LIN {X 0.054,Y -621.065,Z 312.138,A 0.000,B 0.000,C 90.000,E1 240.873} C_DIS
LIN {X 0.084,Y -617.103,Z 312.131,A 0.000,B 0.000,C 90.000,E1 239.587} C_DIS
LIN {X 0.303,Y -613.890,Z 312.125,A 0.000,B 0.000,C 90.000,E1 238.535} C_DIS
LIN {X 0.171,Y -609.063,Z 312.117,A 0.000,B 0.000,C 90.000,E1 236.993} C_DIS
LIN {X 0.075,Y -605.848,Z 312.111,A 0.000,B 0.000,C 90.000,E1 235.960} C_DIS
LIN {X 0.200,Y -600.104,Z 312.101,A 0.000,B 0.000,C 90.000,E1 234.116} C_DIS
LIN {X 0.333,Y -596.624,Z 312.095,A 0.000,B 0.000,C 90.000,E1 233.050} C_DIS
LIN {X -0.237,Y -590.243,Z 312.085,A 0.000,B 0.000,C 90.000,E1 231.251} C_DIS
LIN {X -0.144,Y -585.821,Z 312.077,A 0.000,B 0.000,C 90.000,E1 229.908} C_DIS
LIN {X -0.014,Y -580.499,Z 312.068,A 0.000,B 0.000,C 90.000,E1 228.286} C_DIS
LIN {X -0.102,Y -576.333,Z 312.061,A 0.000,B 0.000,C 90.000,E1 226.944} C_DIS
LIN {X -0.013,Y -572.939,Z 312.055,A 0.000,B 0.000,C 90.000,E1 225.850} C_DIS
LIN {X 0.018,Y -566.044,Z 312.043,A 0.000,B 0.000,C 90.000,E1 223.662} C_DIS
LIN {X 0.033,Y -561.867,Z 312.035,A 0.000,B 0.000,C 90.000,E1 222.285} C_DIS
LIN {X 0.080,Y -556.813,Z 312.026,A 0.000,B 0.000,C 90.000,E1 220.620} C_DIS
LIN {X -0.048,Y -552.562,Z 312.018,A 0.000,B 0.000,C 90.000,E1 219.241} C_DIS
LIN {X -0.129,Y -547.540,Z 312.009,A 0.000,B 0.000,C 90.000,E1 217.569} C_DIS
LIN {X 0.085,Y -543.291,Z 312.001,A 0.000,B 0.000,C 90.000,E1 216.137} C_DIS
LIN {X 0.077,Y -537.670,Z 311.990,A 0.000,B 0.000,C 90.000,E1 214.151} C_DIS
LIN {X -0.197,Y -533.791,Z 311.982,A 0.000,B 0.000,C 90.000,E1 212.752} C_DIS
LIN {X 0.071,Y -529.978,Z 311.974,A 0.000,B 0.000,C 90.000,E1 211.288} C_DIS
LIN {X 0.227,Y -525.621,Z 311.964,A 0.000,B 0.000,C 90.000,E1 209.539} C_DIS
LIN {X 0.147,Y -520.586,Z 311.953,A 0.000,B 0.000,C 90.000,E1 207.513} C_DIS
LIN {X 0.137,Y -517.085,Z 311.945,A 0.000,B 0.000,C 90.000,E1 206.052} C_DIS
LIN {X -0.273,Y -513.125,Z 311.935,A 0.000,B 0.000,C 90.000,E1 204.335} C_DIS
LIN {X 0.154,Y -509.144,Z 311.925,A 0.000,B 0.000,C 90.000,E1 202.514} C_DIS
LIN {X 0.007,Y -506.002,Z 311.917,A 0.000,B 0.000,C 90.000,E1 201.046} C_DIS
LIN {X -0.110,Y -502.294,Z 311.907,A 0.000,B 0.000,C 90.000,E1 199.268} C_DIS
LIN {X 0.051,Y -498.120,Z 311.895,A 0.000,B 0.000,C 90.000,E1 197.149} C_DIS
LIN {X -0.226,Y -494.818,Z 311.885,A 0.000,B 0.000,C 90.000,E1 195.371} C_DIS
LIN {X 0.189,Y -490.358,Z 311.870,A 0.000,B 0.000,C 90.000,E1 192.591} C_DIS
LIN {X -0.109,Y -486.945,Z 311.858,A 0.000,B 0.000,C 90.000,E1 190.489} C_DIS
LIN {X 0.109,Y -484.279,Z 311.848,A 0.000,B 0.000,C 90.000,E1 188.624} C_DIS
LIN {X -0.030,Y -481.304,Z 311.836,A 0.000,B 0.000,C 90.000,E1 186.486} C_DIS
LIN {X 0.219,Y -479.780,Z 311.829,A 0.000,B 0.000,C 90.000,E1 185.220} C_DIS
LIN {X 0.137,Y -476.898,Z 311.815,A 0.000,B 0.000,C 90.000,E1 182.751} C_DIS
LIN {X -0.189,Y -475.590,Z 311.809,A 0.000,B 0.000,C 90.000,E1 181.547} C_DIS
LIN {X -0.126,Y -472.809,Z 311.789,A 0.000,B 0.000,C 90.000,E1 178.108} C_DIS
LIN {X 0.151,Y -471.024,Z 311.769,A 0.000,B 0.000,C 90.000,E1 174.318} C_DIS
LIN {X -0.083,Y -470.413,Z 311.755,A 0.000,B 0.000,C 90.000,E1 171.837} C_DIS
LIN {X 0.080,Y -470.402,Z 311.739,A 0.000,B 0.000,C 90.000,E1 168.993} C_DIS
LIN {X -0.150,Y -470.751,Z 311.727,A 0.000,B 0.000,C 90.000,E1 166.825} C_DIS
LIN {X 0.079,Y -471.940,Z 311.711,A 0.000,B 0.000,C 90.000,E1 163.976} C_DIS
LIN {X -0.195,Y -473.286,Z 311.699,A 0.000,B 0.000,C 90.000,E1 161.819} C_DIS
LIN {X 0.260,Y -475.302,Z 311.683,A 0.000,B 0.000,C 90.000,E1 158.954} C_DIS
LIN {X 0.052,Y -478.623,Z 311.666,A 0.000,B 0.000,C 90.000,E1 155.869} C_DIS
LIN {X 0.114,Y -482.384,Z 311.651,A 0.000,B 0.000,C 90.000,E1 153.076} C_DIS
LIN {X -0.095,Y -486.412,Z 311.637,A 0.000,B 0.000,C 90.000,E1 150.639} C_DIS
LIN {X -0.173,Y -491.133,Z 311.623,A 0.000,B 0.000,C 90.000,E1 148.201} C_DIS
LIN {X 0.279,Y -494.405,Z 311.615,A 0.000,B 0.000,C 90.000,E1 146.628} C_DIS
LIN {X -0.166,Y -499.078,Z 311.603,A 0.000,B 0.000,C 90.000,E1 144.562} C_DIS
LIN {X -0.091,Y -502.259,Z 311.595,A 0.000,B 0.000,C 90.000,E1 143.050} C_DIS
LIN {X 0.049,Y -505.282,Z 311.586,A 0.000,B 0.000,C 90.000,E1 141.537} C_DIS
LIN {X -0.054,Y -507.425,Z 311.580,A 0.000,B 0.000,C 90.000,E1 140.356} C_DIS
LIN {X -0.131,Y -509.353,Z 311.573,A 0.000,B 0.000,C 90.000,E1 139.175} C_DIS
LIN {X 0.247,Y -510.541,Z 311.568,A 0.000,B 0.000,C 90.000,E1 138.243} C_DIS
LIN {X -0.081,Y -511.546,Z 311.563,A 0.000,B 0.000,C 90.000,E1 137.391} C_DIS
LIN {X -0.145,Y -512.482,Z 311.557,A 0.000,B 0.000,C 90.000,E1 136.215} C_DIS
LIN {X 0.161,Y -512.869,Z 311.550,A 0.000,B 0.000,C 90.000,E1 135.000} C_DIS
LIN {X -0.254,Y -512.798,Z 311.544,A 0.000,B 0.000,C 90.000,E1 133.866} C_DIS
LIN {X -0.302,Y -512.292,Z 311.537,A 0.000,B 0.000,C 90.000,E1 132.690} C_DIS
LIN {X 0.113,Y -511.580,Z 311.532,A 0.000,B 0.000,C 90.000,E1 131.757} C_DIS
LIN {X -0.205,Y -510.652,Z 311.527,A 0.000,B 0.000,C 90.000,E1 130.906} C_DIS
LIN {X -0.239,Y -509.147,Z 311.521,A 0.000,B 0.000,C 90.000,E1 129.725} C_DIS
LIN {X -0.071,Y -507.131,Z 311.512,A 0.000,B 0.000,C 90.000,E1 128.222} C_DIS
LIN {X 0.135,Y -505.013,Z 311.504,A 0.000,B 0.000,C 90.000,E1 126.710} C_DIS
LIN {X 0.113,Y -503.165,Z 311.497,A 0.000,B 0.000,C 90.000,E1 125.518} C_DIS
LIN {X -0.055,Y -500.467,Z 311.489,A 0.000,B 0.000,C 90.000,E1 124.040} C_DIS
LIN {X -0.138,Y -497.552,Z 311.481,A 0.000,B 0.000,C 90.000,E1 122.546} C_DIS
LIN {X -0.123,Y -495.184,Z 311.474,A 0.000,B 0.000,C 90.000,E1 121.337} C_DIS
LIN {X 0.118,Y -492.114,Z 311.466,A 0.000,B 0.000,C 90.000,E1 119.795} C_DIS
LIN {X 0.301,Y -487.796,Z 311.454,A 0.000,B 0.000,C 90.000,E1 117.641} C_DIS
LIN {X -0.080,Y -484.713,Z 311.445,A 0.000,B 0.000,C 90.000,E1 116.155} C_DIS
LIN {X 0.143,Y -481.605,Z 311.437,A 0.000,B 0.000,C 90.000,E1 114.591} C_DIS
LIN {X -0.125,Y -478.497,Z 311.428,A 0.000,B 0.000,C 90.000,E1 113.078} C_DIS
LIN {X -0.220,Y -474.768,Z 311.418,A 0.000,B 0.000,C 90.000,E1 111.227} C_DIS
LIN {X 0.038,Y -471.128,Z 311.407,A 0.000,B 0.000,C 90.000,E1 109.322} C_DIS
LIN {X 0.082,Y -466.328,Z 311.393,A 0.000,B 0.000,C 90.000,E1 106.804} C_DIS
LIN {X -0.163,Y -464.954,Z 311.389,A 0.000,B 0.000,C 90.000,E1 106.079} C_DIS
LIN {X -0.202,Y -464.952,Z 311.389,A 0.000,B 0.000,C 90.000,E1 106.079} C_DIS
LIN {X 0.165,Y -467.726,Z 311.383,A 0.000,B 0.000,C 90.000,E1 104.898} C_DIS
LIN {X 0.137,Y -475.934,Z 311.357,A 0.000,B 0.000,C 90.000,E1 100.197} C_DIS
LIN {X -0.024,Y -476.364,Z 311.355,A 0.000,B 0.000,C 90.000,E1 99.905} C_DIS
LIN {X -0.068,Y -481.890,Z 311.331,A 0.000,B 0.000,C 90.000,E1 95.568} C_DIS
LIN {X -0.220,Y -482.197,Z 311.329,A 0.000,B 0.000,C 90.000,E1 95.277} C_DIS
LIN {X 0.198,Y -485.374,Z 311.305,A 0.000,B 0.000,C 90.000,E1 90.917} C_DIS
LIN {X 0.023,Y -485.531,Z 311.304,A 0.000,B 0.000,C 90.000,E1 90.630} C_DIS
LIN {X 0.230,Y -486.350,Z 311.281,A 0.000,B 0.000,C 90.000,E1 86.617} C_DIS
LIN {X 0.055,Y -486.369,Z 311.280,A 0.000,B 0.000,C 90.000,E1 86.331} C_DIS
LIN {X 0.223,Y -486.057,Z 311.276,A 0.000,B 0.000,C 90.000,E1 85.698} C_DIS
LIN {X 0.079,Y -484.693,Z 311.254,A 0.000,B 0.000,C 90.000,E1 81.724} C_DIS
LIN {X -0.053,Y -484.524,Z 311.252,A 0.000,B 0.000,C 90.000,E1 81.432} C_DIS
LIN {X -0.183,Y -480.460,Z 311.227,A 0.000,B 0.000,C 90.000,E1 76.825} C_DIS
LIN {X -0.138,Y -475.986,Z 311.210,A 0.000,B 0.000,C 90.000,E1 73.740} C_DIS
LIN {X 0.178,Y -480.585,Z 311.199,A 0.000,B 0.000,C 90.000,E1 71.819} C_DIS
LIN {X -0.159,Y -485.320,Z 311.189,A 0.000,B 0.000,C 90.000,E1 70.007} C_DIS
LIN {X -0.080,Y -489.458,Z 311.180,A 0.000,B 0.000,C 90.000,E1 68.465} C_DIS
LIN {X 0.044,Y -492.837,Z 311.174,A 0.000,B 0.000,C 90.000,E1 67.230} C_DIS
LIN {X -0.191,Y -497.106,Z 311.165,A 0.000,B 0.000,C 90.000,E1 65.741} C_DIS
LIN {X -0.253,Y -503.092,Z 311.153,A 0.000,B 0.000,C 90.000,E1 63.640} C_DIS
LIN {X 0.123,Y -507.432,Z 311.145,A 0.000,B 0.000,C 90.000,E1 62.103} C_DIS
LIN {X 0.017,Y -512.604,Z 311.135,A 0.000,B 0.000,C 90.000,E1 60.333} C_DIS
LIN {X -0.080,Y -516.937,Z 311.127,A 0.000,B 0.000,C 90.000,E1 58.869} C_DIS
LIN {X -0.162,Y -522.069,Z 311.117,A 0.000,B 0.000,C 90.000,E1 57.120} C_DIS
LIN {X -0.252,Y -526.246,Z 311.109,A 0.000,B 0.000,C 90.000,E1 55.674} C_DIS
LIN {X 0.034,Y -530.220,Z 311.101,A 0.000,B 0.000,C 90.000,E1 54.196} C_DIS
LIN {X -0.023,Y -533.243,Z 311.095,A 0.000,B 0.000,C 90.000,E1 53.050} C_DIS
LIN {X -0.039,Y -535.952,Z 311.088,A 0.000,B 0.000,C 90.000,E1 51.904} C_DIS
LIN {X 0.318,Y -538.475,Z 311.082,A 0.000,B 0.000,C 90.000,E1 50.723} C_DIS
LIN {X -0.077,Y -539.629,Z 311.079,A 0.000,B 0.000,C 90.000,E1 50.194} C_DIS
LIN {X -0.062,Y -542.242,Z 311.071,A 0.000,B 0.000,C 90.000,E1 48.771} C_DIS
LIN {X -0.050,Y -543.727,Z 311.066,A 0.000,B 0.000,C 90.000,E1 47.919} C_DIS
LIN {X -0.022,Y -544.977,Z 311.062,A 0.000,B 0.000,C 90.000,E1 47.067} C_DIS
LIN {X 0.043,Y -546.765,Z 311.054,A 0.000,B 0.000,C 90.000,E1 45.648} C_DIS
LIN {X -0.293,Y -547.576,Z 311.049,A 0.000,B 0.000,C 90.000,E1 44.838} C_DIS
LIN {X 0.194,Y -548.560,Z 311.041,A 0.000,B 0.000,C 90.000,E1 43.380} C_DIS
LIN {X -0.095,Y -549.162,Z 311.035,A 0.000,B 0.000,C 90.000,E1 42.285} C_DIS
LIN {X 0.081,Y -549.559,Z 311.027,A 0.000,B 0.000,C 90.000,E1 40.862} C_DIS
LIN {X 0.168,Y -549.577,Z 311.022,A 0.000,B 0.000,C 90.000,E1 40.011} C_DIS
LIN {X -0.049,Y -549.318,Z 311.016,A 0.000,B 0.000,C 90.000,E1 38.910} C_DIS
LIN {X -0.321,Y -548.907,Z 311.012,A 0.000,B 0.000,C 90.000,E1 38.096} C_DIS
LIN {X -0.063,Y -547.928,Z 311.004,A 0.000,B 0.000,C 90.000,E1 36.664} C_DIS
LIN {X 0.129,Y -546.952,Z 310.997,A 0.000,B 0.000,C 90.000,E1 35.518} C_DIS
LIN {X 0.027,Y -545.669,Z 310.990,A 0.000,B 0.000,C 90.000,E1 34.119} C_DIS
LIN {X 0.056,Y -544.321,Z 310.982,A 0.000,B 0.000,C 90.000,E1 32.704} C_DIS
LIN {X -0.159,Y -542.194,Z 310.969,A 0.000,B 0.000,C 90.000,E1 30.463} C_DIS
LIN {X -0.260,Y -540.386,Z 310.958,A 0.000,B 0.000,C 90.000,E1 28.487} C_DIS
LIN {X -0.111,Y -539.313,Z 310.952,A 0.000,B 0.000,C 90.000,E1 27.334} C_DIS
LIN {X -0.007,Y -537.941,Z 310.944,A 0.000,B 0.000,C 90.000,E1 25.899} C_DIS
LIN {X -0.193,Y -536.382,Z 310.934,A 0.000,B 0.000,C 90.000,E1 24.207} C_DIS
LIN {X -0.199,Y -534.694,Z 310.923,A 0.000,B 0.000,C 90.000,E1 22.206} C_DIS
LIN {X -0.069,Y -533.850,Z 310.917,A 0.000,B 0.000,C 90.000,E1 21.046} C_DIS
LIN {X 0.165,Y -532.393,Z 310.904,A 0.000,B 0.000,C 90.000,E1 18.725} C_DIS
LIN {X 0.189,Y -531.050,Z 310.890,A 0.000,B 0.000,C 90.000,E1 16.134} C_DIS
LIN {X 0.178,Y -530.305,Z 310.879,A 0.000,B 0.000,C 90.000,E1 14.120} C_DIS
LIN {X 0.023,Y -529.791,Z 310.867,A 0.000,B 0.000,C 90.000,E1 12.119} C_DIS
LIN {X 0.202,Y -529.576,Z 310.855,A 0.000,B 0.000,C 90.000,E1 9.792} C_DIS
LIN {X -0.192,Y -529.790,Z 310.840,A 0.000,B 0.000,C 90.000,E1 7.239} C_DIS
LIN {X -0.217,Y -530.398,Z 310.827,A 0.000,B 0.000,C 90.000,E1 4.935} C_DIS
LIN {X -0.264,Y -531.101,Z 310.818,A 0.000,B 0.000,C 90.000,E1 3.212} C_DIS
LIN {X 0.227,Y -532.011,Z 310.808,A 0.000,B 0.000,C 90.000,E1 1.432} C_DIS
LIN {X 0.189,Y -533.352,Z 310.796,A 0.000,B 0.000,C 90.000,E1 359.198} C_DIS
LIN {X 0.175,Y -535.039,Z 310.785,A 0.000,B 0.000,C 90.000,E1 357.192} C_DIS
LIN {X 0.229,Y -536.424,Z 310.777,A 0.000,B 0.000,C 90.000,E1 355.755} C_DIS
LIN {X -0.060,Y -539.508,Z 310.761,A 0.000,B 0.000,C 90.000,E1 352.932} C_DIS
LIN {X 0.205,Y -542.803,Z 310.750,A 0.000,B 0.000,C 90.000,E1 350.914} C_DIS
LIN {X 0.248,Y -549.753,Z 310.731,A 0.000,B 0.000,C 90.000,E1 347.521} C_DIS
LIN {X -0.151,Y -554.083,Z 310.722,A 0.000,B 0.000,C 90.000,E1 345.880} C_DIS
LIN {X 0.231,Y -560.124,Z 310.709,A 0.000,B 0.000,C 90.000,E1 343.614} C_DIS
LIN {X -0.212,Y -564.870,Z 310.700,A 0.000,B 0.000,C 90.000,E1 342.000} C_DIS
LIN {X 0.143,Y -569.679,Z 310.691,A 0.000,B 0.000,C 90.000,E1 340.315} C_DIS
LIN {X 0.299,Y -571.368,Z 310.688,A 0.000,B 0.000,C 90.000,E1 339.752} C_DIS
LIN {X 0.095,Y -573.791,Z 310.683,A 0.000,B 0.000,C 90.000,E1 338.954} C_DIS
LIN {X 0.291,Y -577.312,Z 310.677,A 0.000,B 0.000,C 90.000,E1 337.847} C_DIS
LIN {X -0.002,Y -580.918,Z 310.671,A 0.000,B 0.000,C 90.000,E1 336.794} C_DIS
LIN {X 0.148,Y -585.383,Z 310.664,A 0.000,B 0.000,C 90.000,E1 335.433} C_DIS
LIN {X -0.135,Y -592.066,Z 310.653,A 0.000,B 0.000,C 90.000,E1 333.589} C_DIS
LIN {X 0.092,Y -597.745,Z 310.644,A 0.000,B 0.000,C 90.000,E1 331.975} C_DIS
LIN {X -0.018,Y -602.312,Z 310.637,A 0.000,B 0.000,C 90.000,E1 330.667} C_DIS
LIN {X 0.192,Y -607.892,Z 310.628,A 0.000,B 0.000,C 90.000,E1 329.076} C_DIS
LIN {X 0.278,Y -614.299,Z 310.618,A 0.000,B 0.000,C 90.000,E1 327.248} C_DIS
LIN {X 0.273,Y -617.854,Z 310.612,A 0.000,B 0.000,C 90.000,E1 326.215} C_DIS
LIN {X -0.228,Y -622.276,Z 310.605,A 0.000,B 0.000,C 90.000,E1 324.975} C_DIS
LIN {X -0.110,Y -624.819,Z 310.601,A 0.000,B 0.000,C 90.000,E1 324.196} C_DIS
LIN {X 0.386,Y -628.014,Z 310.595,A 0.000,B 0.000,C 90.000,E1 323.130} C_DIS
LIN {X -0.099,Y -631.744,Z 310.588,A 0.000,B 0.000,C 90.000,E1 321.904} C_DIS
LIN {X 0.246,Y -636.116,Z 310.580,A 0.000,B 0.000,C 90.000,E1 320.356} C_DIS
LIN {X 0.193,Y -640.561,Z 310.572,A 0.000,B 0.000,C 90.000,E1 318.852} C_DIS
LIN {X -0.103,Y -643.426,Z 310.566,A 0.000,B 0.000,C 90.000,E1 317.877} C_DIS
LIN {X -0.308,Y -650.814,Z 310.552,A 0.000,B 0.000,C 90.000,E1 315.405} C_DIS
LIN {X -0.047,Y -653.782,Z 310.547,A 0.000,B 0.000,C 90.000,E1 314.393} C_DIS
LIN {X -0.225,Y -657.191,Z 310.540,A 0.000,B 0.000,C 90.000,E1 313.176} C_DIS
LIN {X 0.113,Y -660.442,Z 310.533,A 0.000,B 0.000,C 90.000,E1 311.919} C_DIS
LIN {X -0.398,Y -662.295,Z 310.529,A 0.000,B 0.000,C 90.000,E1 311.229} C_DIS
LIN {X 0.022,Y -664.597,Z 310.523,A 0.000,B 0.000,C 90.000,E1 310.216} C_DIS
LIN {X 0.115,Y -667.184,Z 310.517,A 0.000,B 0.000,C 90.000,E1 308.991} C_DIS
LIN {X 0.165,Y -669.104,Z 310.511,A 0.000,B 0.000,C 90.000,E1 308.016} C_DIS
LIN {X -0.165,Y -670.398,Z 310.507,A 0.000,B 0.000,C 90.000,E1 307.317} C_DIS
LIN {X -0.093,Y -671.847,Z 310.502,A 0.000,B 0.000,C 90.000,E1 306.343} C_DIS
LIN {X -0.258,Y -673.002,Z 310.497,A 0.000,B 0.000,C 90.000,E1 305.391} C_DIS
LIN {X 0.396,Y -673.569,Z 310.493,A 0.000,B 0.000,C 90.000,E1 304.612} C_DIS
LIN {X 0.113,Y -673.892,Z 310.488,A 0.000,B 0.000,C 90.000,E1 303.913} C_DIS
LIN {X -0.009,Y -673.873,Z 310.483,A 0.000,B 0.000,C 90.000,E1 302.959} C_DIS
LIN {X 0.275,Y -673.725,Z 310.479,A 0.000,B 0.000,C 90.000,E1 302.212} C_DIS
LIN {X -0.019,Y -673.187,Z 310.475,A 0.000,B 0.000,C 90.000,E1 301.514} C_DIS
LIN {X -0.096,Y -672.317,Z 310.471,A 0.000,B 0.000,C 90.000,E1 300.797} C_DIS
LIN {X 0.328,Y -670.772,Z 310.466,A 0.000,B 0.000,C 90.000,E1 299.795} C_DIS
LIN {X 0.236,Y -669.265,Z 310.462,A 0.000,B 0.000,C 90.000,E1 299.077} C_DIS
LIN {X -0.143,Y -666.552,Z 310.455,A 0.000,B 0.000,C 90.000,E1 297.897} C_DIS
LIN {X 0.016,Y -663.590,Z 310.448,A 0.000,B 0.000,C 90.000,E1 296.668} C_DIS
LIN {X -0.167,Y -660.470,Z 310.441,A 0.000,B 0.000,C 90.000,E1 295.463} C_DIS
LIN {X 0.198,Y -657.146,Z 310.435,A 0.000,B 0.000,C 90.000,E1 294.207} C_DIS
LIN {X -0.243,Y -653.100,Z 310.426,A 0.000,B 0.000,C 90.000,E1 292.770} C_DIS
LIN {X -0.194,Y -651.088,Z 310.422,A 0.000,B 0.000,C 90.000,E1 292.025} C_DIS
LIN {X -0.163,Y -647.115,Z 310.414,A 0.000,B 0.000,C 90.000,E1 290.536} C_DIS
LIN {X -0.164,Y -642.085,Z 310.403,A 0.000,B 0.000,C 90.000,E1 288.544} C_DIS
LIN {X -0.197,Y -635.149,Z 310.386,A 0.000,B 0.000,C 90.000,E1 285.536} C_DIS
LIN {X -0.172,Y -630.235,Z 310.372,A 0.000,B 0.000,C 90.000,E1 283.008} C_DIS
LIN {X -0.215,Y -625.615,Z 310.355,A 0.000,B 0.000,C 90.000,E1 279.962} C_DIS
LIN {X 0.000,Y -622.967,Z 310.343,A 0.000,B 0.000,C 90.000,E1 277.644} C_DIS
LIN {X 0.053,Y -621.061,Z 310.330,A 0.000,B 0.000,C 90.000,E1 275.334} C_DIS
LIN {X 0.244,Y -619.846,Z 310.315,A 0.000,B 0.000,C 90.000,E1 272.751} C_DIS
LIN {X 0.052,Y -619.395,Z 310.300,A 0.000,B 0.000,C 90.000,E1 269.943} C_DIS
LIN {X 0.173,Y -620.108,Z 310.283,A 0.000,B 0.000,C 90.000,E1 266.849} C_DIS
LIN {X -0.271,Y -621.277,Z 310.271,A 0.000,B 0.000,C 90.000,E1 264.837} C_DIS
LIN {X 0.007,Y -622.958,Z 310.260,A 0.000,B 0.000,C 90.000,E1 262.761} C_DIS
LIN {X 0.195,Y -625.348,Z 310.247,A 0.000,B 0.000,C 90.000,E1 260.443} C_DIS
LIN {X 0.145,Y -627.977,Z 310.236,A 0.000,B 0.000,C 90.000,E1 258.409} C_DIS
LIN {X -0.201,Y -630.937,Z 310.224,A 0.000,B 0.000,C 90.000,E1 256.408} C_DIS
LIN {X 0.058,Y -633.131,Z 310.216,A 0.000,B 0.000,C 90.000,E1 254.866} C_DIS
LIN {X 0.302,Y -633.774,Z 310.213,A 0.000,B 0.000,C 90.000,E1 254.338} C_DIS
LIN {X 0.178,Y -634.938,Z 310.206,A 0.000,B 0.000,C 90.000,E1 253.087} C_DIS
LIN {X -0.360,Y -635.842,Z 310.201,A 0.000,B 0.000,C 90.000,E1 252.127} C_DIS
LIN {X -0.082,Y -636.461,Z 310.195,A 0.000,B 0.000,C 90.000,E1 251.094} C_DIS
LIN {X 0.178,Y -636.676,Z 310.191,A 0.000,B 0.000,C 90.000,E1 250.315} C_DIS
LIN {X -0.133,Y -636.627,Z 310.185,A 0.000,B 0.000,C 90.000,E1 249.337} C_DIS
LIN {X -0.251,Y -636.412,Z 310.181,A 0.000,B 0.000,C 90.000,E1 248.592} C_DIS
LIN {X 0.263,Y -635.595,Z 310.175,A 0.000,B 0.000,C 90.000,E1 247.539} C_DIS
LIN {X 0.098,Y -635.033,Z 310.173,A 0.000,B 0.000,C 90.000,E1 247.050} C_DIS
LIN {X 0.181,Y -634.369,Z 310.170,A 0.000,B 0.000,C 90.000,E1 246.538} C_DIS
LIN {X 0.045,Y -633.128,Z 310.166,A 0.000,B 0.000,C 90.000,E1 245.793} C_DIS
LIN {X 0.121,Y -632.218,Z 310.163,A 0.000,B 0.000,C 90.000,E1 245.281} C_DIS
LIN {X -0.043,Y -630.586,Z 310.159,A 0.000,B 0.000,C 90.000,E1 244.537} C_DIS
LIN {X 0.071,Y -628.088,Z 310.153,A 0.000,B 0.000,C 90.000,E1 243.512} C_DIS
LIN {X 0.151,Y -625.236,Z 310.147,A 0.000,B 0.000,C 90.000,E1 242.487} C_DIS
LIN {X -0.358,Y -621.437,Z 310.140,A 0.000,B 0.000,C 90.000,E1 241.257} C_DIS
LIN {X -0.093,Y -617.580,Z 310.133,A 0.000,B 0.000,C 90.000,E1 239.950} C_DIS
LIN {X -0.114,Y -613.641,Z 310.126,A 0.000,B 0.000,C 90.000,E1 238.663} C_DIS
LIN {X -0.243,Y -608.795,Z 310.117,A 0.000,B 0.000,C 90.000,E1 237.120} C_DIS
LIN {X -0.337,Y -605.632,Z 310.111,A 0.000,B 0.000,C 90.000,E1 236.087} C_DIS
LIN {X -0.221,Y -601.541,Z 310.104,A 0.000,B 0.000,C 90.000,E1 234.769} C_DIS
LIN {X -0.313,Y -599.112,Z 310.100,A 0.000,B 0.000,C 90.000,E1 233.989} C_DIS
LIN {X -0.194,Y -595.564,Z 310.094,A 0.000,B 0.000,C 90.000,E1 232.924} C_DIS
LIN {X 0.037,Y -589.256,Z 310.084,A 0.000,B 0.000,C 90.000,E1 231.045} C_DIS
LIN {X 0.106,Y -584.857,Z 310.076,A 0.000,B 0.000,C 90.000,E1 229.703} C_DIS
LIN {X 0.208,Y -579.597,Z 310.067,A 0.000,B 0.000,C 90.000,E1 228.081} C_DIS
LIN {X 0.068,Y -575.454,Z 310.060,A 0.000,B 0.000,C 90.000,E1 226.743} C_DIS
LIN {X 0.152,Y -572.042,Z 310.054,A 0.000,B 0.000,C 90.000,E1 225.648} C_DIS
LIN {X -0.335,Y -566.078,Z 310.043,A 0.000,B 0.000,C 90.000,E1 223.785} C_DIS
LIN {X 0.090,Y -561.927,Z 310.035,A 0.000,B 0.000,C 90.000,E1 222.366} C_DIS
LIN {X 0.058,Y -557.749,Z 310.028,A 0.000,B 0.000,C 90.000,E1 220.987} C_DIS
LIN {X 0.020,Y -553.531,Z 310.020,A 0.000,B 0.000,C 90.000,E1 219.600} C_DIS
LIN {X -0.114,Y -548.496,Z 310.011,A 0.000,B 0.000,C 90.000,E1 217.935} C_DIS
LIN {X 0.119,Y -544.254,Z 310.003,A 0.000,B 0.000,C 90.000,E1 216.503} C_DIS
LIN {X 0.011,Y -537.756,Z 309.990,A 0.000,B 0.000,C 90.000,E1 214.246} C_DIS
LIN {X 0.180,Y -534.636,Z 309.984,A 0.000,B 0.000,C 90.000,E1 213.086} C_DIS
LIN {X 0.131,Y -529.207,Z 309.973,A 0.000,B 0.000,C 90.000,E1 211.082} C_DIS
LIN {X 0.265,Y -524.860,Z 309.963,A 0.000,B 0.000,C 90.000,E1 209.333} C_DIS
LIN {X -0.079,Y -519.798,Z 309.952,A 0.000,B 0.000,C 90.000,E1 207.334} C_DIS
LIN {X 0.131,Y -516.279,Z 309.944,A 0.000,B 0.000,C 90.000,E1 205.848} C_DIS
LIN {X 0.043,Y -513.004,Z 309.936,A 0.000,B 0.000,C 90.000,E1 204.387} C_DIS
LIN {X -0.100,Y -508.399,Z 309.924,A 0.000,B 0.000,C 90.000,E1 202.333} C_DIS
LIN {X -0.163,Y -504.665,Z 309.914,A 0.000,B 0.000,C 90.000,E1 200.556} C_DIS
LIN {X 0.089,Y -501.654,Z 309.906,A 0.000,B 0.000,C 90.000,E1 199.033} C_DIS
LIN {X 0.238,Y -497.600,Z 309.894,A 0.000,B 0.000,C 90.000,E1 196.913} C_DIS
LIN {X -0.196,Y -492.370,Z 309.877,A 0.000,B 0.000,C 90.000,E1 193.939} C_DIS
LIN {X -0.129,Y -489.983,Z 309.869,A 0.000,B 0.000,C 90.000,E1 192.411} C_DIS
LIN {X 0.038,Y -486.615,Z 309.857,A 0.000,B 0.000,C 90.000,E1 190.254} C_DIS
LIN {X -0.178,Y -484.454,Z 309.849,A 0.000,B 0.000,C 90.000,E1 188.746} C_DIS
LIN {X 0.182,Y -481.486,Z 309.837,A 0.000,B 0.000,C 90.000,E1 186.549} C_DIS
LIN {X -0.192,Y -479.552,Z 309.828,A 0.000,B 0.000,C 90.000,E1 185.049} C_DIS
LIN {X 0.202,Y -476.726,Z 309.814,A 0.000,B 0.000,C 90.000,E1 182.522} C_DIS
LIN {X -0.126,Y -475.405,Z 309.807,A 0.000,B 0.000,C 90.000,E1 181.318} C_DIS
LIN {X 0.148,Y -472.962,Z 309.790,A 0.000,B 0.000,C 90.000,E1 178.165} C_DIS
LIN {X 0.151,Y -471.273,Z 309.771,A 0.000,B 0.000,C 90.000,E1 174.723} C_DIS
LIN {X -0.080,Y -470.643,Z 309.757,A 0.000,B 0.000,C 90.000,E1 172.243} C_DIS
LIN {X -0.084,Y -470.520,Z 309.739,A 0.000,B 0.000,C 90.000,E1 169.106} C_DIS
LIN {X 0.188,Y -471.119,Z 309.722,A 0.000,B 0.000,C 90.000,E1 165.936} C_DIS
LIN {X 0.212,Y -472.148,Z 309.710,A 0.000,B 0.000,C 90.000,E1 163.740} C_DIS
LIN {X -0.061,Y -473.472,Z 309.698,A 0.000,B 0.000,C 90.000,E1 161.583} C_DIS
LIN {X 0.001,Y -475.046,Z 309.686,A 0.000,B 0.000,C 90.000,E1 159.390} C_DIS
LIN {X -0.142,Y -476.710,Z 309.675,A 0.000,B 0.000,C 90.000,E1 157.539} C_DIS
LIN {X -0.044,Y -478.543,Z 309.667,A 0.000,B 0.000,C 90.000,E1 155.973} C_DIS
LIN {X 0.033,Y -482.245,Z 309.651,A 0.000,B 0.000,C 90.000,E1 153.179} C_DIS
LIN {X 0.024,Y -486.208,Z 309.637,A 0.000,B 0.000,C 90.000,E1 150.717} C_DIS
LIN {X -0.234,Y -491.462,Z 309.622,A 0.000,B 0.000,C 90.000,E1 147.995} C_DIS
LIN {X 0.225,Y -494.635,Z 309.614,A 0.000,B 0.000,C 90.000,E1 146.421} C_DIS
LIN {X 0.073,Y -499.143,Z 309.602,A 0.000,B 0.000,C 90.000,E1 144.322} C_DIS
LIN {X -0.023,Y -501.622,Z 309.595,A 0.000,B 0.000,C 90.000,E1 143.130} C_DIS
LIN {X 0.103,Y -504.588,Z 309.587,A 0.000,B 0.000,C 90.000,E1 141.618} C_DIS
LIN {X -0.013,Y -506.685,Z 309.580,A 0.000,B 0.000,C 90.000,E1 140.436} C_DIS
LIN {X -0.101,Y -508.590,Z 309.574,A 0.000,B 0.000,C 90.000,E1 139.256} C_DIS
LIN {X 0.266,Y -509.757,Z 309.569,A 0.000,B 0.000,C 90.000,E1 138.324} C_DIS
LIN {X -0.069,Y -510.762,Z 309.564,A 0.000,B 0.000,C 90.000,E1 137.472} C_DIS
LIN {X -0.045,Y -511.443,Z 309.559,A 0.000,B 0.000,C 90.000,E1 136.581} C_DIS
LIN {X 0.107,Y -511.858,Z 309.556,A 0.000,B 0.000,C 90.000,E1 135.972} C_DIS
LIN {X 0.040,Y -512.129,Z 309.549,A 0.000,B 0.000,C 90.000,E1 134.798} C_DIS
LIN {X -0.279,Y -512.055,Z 309.544,A 0.000,B 0.000,C 90.000,E1 133.947} C_DIS
LIN {X 0.134,Y -511.735,Z 309.539,A 0.000,B 0.000,C 90.000,E1 133.014} C_DIS
LIN {X -0.179,Y -511.122,Z 309.534,A 0.000,B 0.000,C 90.000,E1 132.162} C_DIS
LIN {X 0.223,Y -510.290,Z 309.529,A 0.000,B 0.000,C 90.000,E1 131.229} C_DIS
LIN {X 0.028,Y -508.518,Z 309.521,A 0.000,B 0.000,C 90.000,E1 129.769} C_DIS
LIN {X -0.239,Y -506.074,Z 309.511,A 0.000,B 0.000,C 90.000,E1 128.016} C_DIS
LIN {X 0.057,Y -504.360,Z 309.504,A 0.000,B 0.000,C 90.000,E1 126.790} C_DIS
LIN {X 0.029,Y -502.503,Z 309.498,A 0.000,B 0.000,C 90.000,E1 125.598} C_DIS
LIN {X -0.025,Y -500.364,Z 309.491,A 0.000,B 0.000,C 90.000,E1 124.405} C_DIS
LIN {X -0.116,Y -498.114,Z 309.484,A 0.000,B 0.000,C 90.000,E1 123.214} C_DIS
LIN {X 0.029,Y -494.589,Z 309.474,A 0.000,B 0.000,C 90.000,E1 121.386} C_DIS
LIN {X 0.264,Y -490.887,Z 309.464,A 0.000,B 0.000,C 90.000,E1 119.539} C_DIS
LIN {X 0.182,Y -487.208,Z 309.454,A 0.000,B 0.000,C 90.000,E1 117.719} C_DIS
LIN {X -0.204,Y -484.118,Z 309.446,A 0.000,B 0.000,C 90.000,E1 116.232} C_DIS
LIN {X 0.215,Y -481.035,Z 309.437,A 0.000,B 0.000,C 90.000,E1 114.643} C_DIS
LIN {X -0.083,Y -477.301,Z 309.427,A 0.000,B 0.000,C 90.000,E1 112.823} C_DIS
LIN {X -0.158,Y -474.876,Z 309.420,A 0.000,B 0.000,C 90.000,E1 111.589} C_DIS
LIN {X -0.059,Y -471.233,Z 309.409,A 0.000,B 0.000,C 90.000,E1 109.704} C_DIS
LIN {X -0.043,Y -467.597,Z 309.399,A 0.000,B 0.000,C 90.000,E1 107.819} C_DIS
LIN {X -0.265,Y -464.685,Z 309.390,A 0.000,B 0.000,C 90.000,E1 106.205} C_DIS
LIN {X 0.142,Y -464.687,Z 309.390,A 0.000,B 0.000,C 90.000,E1 106.150} C_DIS
LIN {X 0.152,Y -467.594,Z 309.383,A 0.000,B 0.000,C 90.000,E1 104.954} C_DIS
LIN {X -0.115,Y -468.592,Z 309.380,A 0.000,B 0.000,C 90.000,E1 104.356} C_DIS
LIN {X 0.111,Y -475.823,Z 309.357,A 0.000,B 0.000,C 90.000,E1 100.254} C_DIS
LIN {X -0.052,Y -476.314,Z 309.355,A 0.000,B 0.000,C 90.000,E1 99.962} C_DIS
LIN {X -0.104,Y -481.805,Z 309.331,A 0.000,B 0.000,C 90.000,E1 95.625} C_DIS
LIN {X 0.222,Y -482.175,Z 309.330,A 0.000,B 0.000,C 90.000,E1 95.277} C_DIS
LIN {X 0.157,Y -485.319,Z 309.306,A 0.000,B 0.000,C 90.000,E1 90.974} C_DIS
LIN {X -0.018,Y -485.536,Z 309.304,A 0.000,B 0.000,C 90.000,E1 90.688} C_DIS
LIN {X 0.189,Y -486.324,Z 309.282,A 0.000,B 0.000,C 90.000,E1 86.674} C_DIS
LIN {X -0.161,Y -486.298,Z 309.278,A 0.000,B 0.000,C 90.000,E1 86.102} C_DIS
LIN {X 0.043,Y -484.695,Z 309.254,A 0.000,B 0.000,C 90.000,E1 81.781} C_DIS
LIN {X -0.089,Y -484.588,Z 309.253,A 0.000,B 0.000,C 90.000,E1 81.489} C_DIS
LIN {X -0.209,Y -480.524,Z 309.227,A 0.000,B 0.000,C 90.000,E1 76.881} C_DIS
LIN {X -0.132,Y -475.792,Z 309.209,A 0.000,B 0.000,C 90.000,E1 73.559} C_DIS
LIN {X -0.023,Y -481.353,Z 309.196,A 0.000,B 0.000,C 90.000,E1 71.275} C_DIS
LIN {X -0.129,Y -488.603,Z 309.181,A 0.000,B 0.000,C 90.000,E1 68.518} C_DIS
LIN {X 0.021,Y -492.802,Z 309.172,A 0.000,B 0.000,C 90.000,E1 66.975} C_DIS
LIN {X -0.212,Y -497.069,Z 309.164,A 0.000,B 0.000,C 90.000,E1 65.485} C_DIS
LIN {X -0.273,Y -503.050,Z 309.152,A 0.000,B 0.000,C 90.000,E1 63.384} C_DIS
LIN {X 0.025,Y -506.550,Z 309.145,A 0.000,B 0.000,C 90.000,E1 62.153} C_DIS
LIN {X -0.094,Y -511.730,Z 309.135,A 0.000,B 0.000,C 90.000,E1 60.383} C_DIS
LIN {X 0.242,Y -516.076,Z 309.127,A 0.000,B 0.000,C 90.000,E1 58.869} C_DIS
LIN {X -0.234,Y -520.331,Z 309.119,A 0.000,B 0.000,C 90.000,E1 57.454} C_DIS
LIN {X 0.039,Y -525.419,Z 309.109,A 0.000,B 0.000,C 90.000,E1 55.674} C_DIS
LIN {X 0.312,Y -529.405,Z 309.101,A 0.000,B 0.000,C 90.000,E1 54.196} C_DIS
LIN {X 0.245,Y -532.411,Z 309.095,A 0.000,B 0.000,C 90.000,E1 53.050} C_DIS
LIN {X 0.219,Y -535.126,Z 309.089,A 0.000,B 0.000,C 90.000,E1 51.904} C_DIS
LIN {X -0.193,Y -537.684,Z 309.082,A 0.000,B 0.000,C 90.000,E1 50.803} C_DIS
LIN {X -0.216,Y -540.451,Z 309.074,A 0.000,B 0.000,C 90.000,E1 49.380} C_DIS
LIN {X 0.170,Y -542.928,Z 309.066,A 0.000,B 0.000,C 90.000,E1 47.919} C_DIS
LIN {X 0.190,Y -544.258,Z 309.062,A 0.000,B 0.000,C 90.000,E1 47.067} C_DIS
LIN {X 0.242,Y -546.007,Z 309.054,A 0.000,B 0.000,C 90.000,E1 45.648} C_DIS
LIN {X 0.270,Y -546.590,Z 309.051,A 0.000,B 0.000,C 90.000,E1 45.081} C_DIS
LIN {X 0.338,Y -547.446,Z 309.044,A 0.000,B 0.000,C 90.000,E1 43.947} C_DIS
LIN {X 0.035,Y -548.181,Z 309.038,A 0.000,B 0.000,C 90.000,E1 42.852} C_DIS
LIN {X -0.256,Y -548.609,Z 309.032,A 0.000,B 0.000,C 90.000,E1 41.757} C_DIS
LIN {X -0.133,Y -548.873,Z 309.026,A 0.000,B 0.000,C 90.000,E1 40.620} C_DIS
LIN {X -0.011,Y -548.826,Z 309.019,A 0.000,B 0.000,C 90.000,E1 39.483} C_DIS
LIN {X 0.139,Y -548.587,Z 309.015,A 0.000,B 0.000,C 90.000,E1 38.624} C_DIS
LIN {X -0.140,Y -548.140,Z 309.010,A 0.000,B 0.000,C 90.000,E1 37.810} C_DIS
LIN {X 0.057,Y -547.373,Z 309.004,A 0.000,B 0.000,C 90.000,E1 36.664} C_DIS
LIN {X 0.240,Y -546.447,Z 308.997,A 0.000,B 0.000,C 90.000,E1 35.518} C_DIS
LIN {X -0.139,Y -544.929,Z 308.988,A 0.000,B 0.000,C 90.000,E1 33.865} C_DIS
LIN {X 0.177,Y -543.566,Z 308.980,A 0.000,B 0.000,C 90.000,E1 32.418} C_DIS
LIN {X -0.071,Y -541.469,Z 308.968,A 0.000,B 0.000,C 90.000,E1 30.178} C_DIS
LIN {X 0.018,Y -539.641,Z 308.957,A 0.000,B 0.000,C 90.000,E1 28.180} C_DIS
LIN {X -0.133,Y -538.024,Z 308.947,A 0.000,B 0.000,C 90.000,E1 26.488} C_DIS
LIN {X -0.152,Y -535.879,Z 308.934,A 0.000,B 0.000,C 90.000,E1 24.207} C_DIS
LIN {X 0.236,Y -533.766,Z 308.920,A 0.000,B 0.000,C 90.000,E1 21.589} C_DIS
LIN {X 0.167,Y -531.818,Z 308.904,A 0.000,B 0.000,C 90.000,E1 18.725} C_DIS
LIN {X 0.201,Y -530.306,Z 308.888,A 0.000,B 0.000,C 90.000,E1 15.843} C_DIS
LIN {X -0.272,Y -529.383,Z 308.874,A 0.000,B 0.000,C 90.000,E1 13.300} C_DIS
LIN {X 0.038,Y -529.044,Z 308.864,A 0.000,B 0.000,C 90.000,E1 11.535} C_DIS
LIN {X 0.133,Y -528.857,Z 308.855,A 0.000,B 0.000,C 90.000,E1 9.792} C_DIS
LIN {X 0.253,Y -528.859,Z 308.848,A 0.000,B 0.000,C 90.000,E1 8.624} C_DIS
LIN {X 0.227,Y -529.119,Z 308.837,A 0.000,B 0.000,C 90.000,E1 6.606} C_DIS
LIN {X 0.213,Y -529.672,Z 308.826,A 0.000,B 0.000,C 90.000,E1 4.588} C_DIS
LIN {X 0.132,Y -530.235,Z 308.818,A 0.000,B 0.000,C 90.000,E1 3.154} C_DIS
LIN {X 0.090,Y -530.954,Z 308.810,A 0.000,B 0.000,C 90.000,E1 1.718} C_DIS
LIN {X 0.201,Y -532.028,Z 308.799,A 0.000,B 0.000,C 90.000,E1 359.771} C_DIS
LIN {X 0.150,Y -533.853,Z 308.786,A 0.000,B 0.000,C 90.000,E1 357.478} C_DIS
LIN {X 0.180,Y -535.455,Z 308.777,A 0.000,B 0.000,C 90.000,E1 355.755} C_DIS
LIN {X -0.246,Y -537.451,Z 308.765,A 0.000,B 0.000,C 90.000,E1 353.799} C_DIS
LIN {X -0.038,Y -544.392,Z 308.742,A 0.000,B 0.000,C 90.000,E1 349.511} C_DIS
LIN {X -0.127,Y -550.829,Z 308.726,A 0.000,B 0.000,C 90.000,E1 346.700} C_DIS
LIN {X -0.255,Y -555.932,Z 308.715,A 0.000,B 0.000,C 90.000,E1 344.755} C_DIS
LIN {X 0.148,Y -559.787,Z 308.707,A 0.000,B 0.000,C 90.000,E1 343.323} C_DIS
LIN {X 0.006,Y -565.306,Z 308.697,A 0.000,B 0.000,C 90.000,E1 341.402} C_DIS
LIN {X 0.025,Y -570.219,Z 308.688,A 0.000,B 0.000,C 90.000,E1 339.752} C_DIS
LIN {X -0.192,Y -572.679,Z 308.683,A 0.000,B 0.000,C 90.000,E1 338.954} C_DIS
LIN {X -0.174,Y -578.923,Z 308.672,A 0.000,B 0.000,C 90.000,E1 337.050} C_DIS
LIN {X 0.047,Y -584.291,Z 308.663,A 0.000,B 0.000,C 90.000,E1 335.409} C_DIS
LIN {X 0.282,Y -590.983,Z 308.653,A 0.000,B 0.000,C 90.000,E1 333.512} C_DIS
LIN {X -0.028,Y -596.652,Z 308.644,A 0.000,B 0.000,C 90.000,E1 331.948} C_DIS
LIN {X 0.379,Y -601.198,Z 308.637,A 0.000,B 0.000,C 90.000,E1 330.589} C_DIS
LIN {X -0.256,Y -606.757,Z 308.628,A 0.000,B 0.000,C 90.000,E1 329.076} C_DIS
LIN {X 0.082,Y -614.068,Z 308.617,A 0.000,B 0.000,C 90.000,E1 326.962} C_DIS
LIN {X 0.344,Y -619.438,Z 308.608,A 0.000,B 0.000,C 90.000,E1 325.388} C_DIS
LIN {X -0.104,Y -622.974,Z 308.602,A 0.000,B 0.000,C 90.000,E1 324.402} C_DIS
LIN {X -0.007,Y -626.261,Z 308.597,A 0.000,B 0.000,C 90.000,E1 323.371} C_DIS
LIN {X -0.001,Y -629.322,Z 308.591,A 0.000,B 0.000,C 90.000,E1 322.351} C_DIS
LIN {X -0.077,Y -632.994,Z 308.584,A 0.000,B 0.000,C 90.000,E1 321.090} C_DIS
LIN {X 0.191,Y -638.208,Z 308.574,A 0.000,B 0.000,C 90.000,E1 319.299} C_DIS
LIN {X -0.131,Y -641.147,Z 308.568,A 0.000,B 0.000,C 90.000,E1 318.324} C_DIS
LIN {X 0.062,Y -648.362,Z 308.555,A 0.000,B 0.000,C 90.000,E1 315.810} C_DIS
LIN {X -0.216,Y -652.128,Z 308.548,A 0.000,B 0.000,C 90.000,E1 314.595} C_DIS
LIN {X 0.037,Y -655.585,Z 308.541,A 0.000,B 0.000,C 90.000,E1 313.338} C_DIS
LIN {X -0.137,Y -658.857,Z 308.534,A 0.000,B 0.000,C 90.000,E1 312.123} C_DIS
LIN {X -0.171,Y -660.741,Z 308.530,A 0.000,B 0.000,C 90.000,E1 311.391} C_DIS
LIN {X 0.231,Y -663.086,Z 308.524,A 0.000,B 0.000,C 90.000,E1 310.378} C_DIS
LIN {X -0.213,Y -665.689,Z 308.518,A 0.000,B 0.000,C 90.000,E1 309.197} C_DIS
LIN {X 0.338,Y -667.593,Z 308.512,A 0.000,B 0.000,C 90.000,E1 308.177} C_DIS
LIN {X 0.403,Y -668.929,Z 308.508,A 0.000,B 0.000,C 90.000,E1 307.443} C_DIS
LIN {X 0.076,Y -670.067,Z 308.504,A 0.000,B 0.000,C 90.000,E1 306.744} C_DIS
LIN {X -0.256,Y -671.366,Z 308.499,A 0.000,B 0.000,C 90.000,E1 305.804} C_DIS
LIN {X 0.379,Y -672.037,Z 308.495,A 0.000,B 0.000,C 90.000,E1 305.025} C_DIS
LIN {X 0.112,Y -672.351,Z 308.492,A 0.000,B 0.000,C 90.000,E1 304.565} C_DIS
LIN {X -0.177,Y -672.638,Z 308.488,A 0.000,B 0.000,C 90.000,E1 303.865} C_DIS
LIN {X 0.056,Y -672.632,Z 308.483,A 0.000,B 0.000,C 90.000,E1 302.880} C_DIS
LIN {X 0.324,Y -672.422,Z 308.479,A 0.000,B 0.000,C 90.000,E1 302.133} C_DIS
LIN {X 0.075,Y -672.090,Z 308.476,A 0.000,B 0.000,C 90.000,E1 301.671} C_DIS
LIN {X -0.077,Y -670.932,Z 308.471,A 0.000,B 0.000,C 90.000,E1 300.718} C_DIS
LIN {X -0.170,Y -669.724,Z 308.467,A 0.000,B 0.000,C 90.000,E1 300.001} C_DIS
LIN {X -0.269,Y -668.310,Z 308.463,A 0.000,B 0.000,C 90.000,E1 299.283} C_DIS
LIN {X 0.244,Y -665.593,Z 308.456,A 0.000,B 0.000,C 90.000,E1 298.025} C_DIS
LIN {X 0.087,Y -662.628,Z 308.449,A 0.000,B 0.000,C 90.000,E1 296.821} C_DIS
LIN {X 0.186,Y -659.542,Z 308.442,A 0.000,B 0.000,C 90.000,E1 295.591} C_DIS
LIN {X 0.054,Y -655.572,Z 308.434,A 0.000,B 0.000,C 90.000,E1 294.131} C_DIS
LIN {X 0.022,Y -650.852,Z 308.425,A 0.000,B 0.000,C 90.000,E1 292.408} C_DIS
LIN {X 0.131,Y -646.198,Z 308.415,A 0.000,B 0.000,C 90.000,E1 290.663} C_DIS
LIN {X 0.148,Y -640.492,Z 308.402,A 0.000,B 0.000,C 90.000,E1 288.417} C_DIS
LIN {X 0.048,Y -634.148,Z 308.387,A 0.000,B 0.000,C 90.000,E1 285.662} C_DIS
LIN {X -0.002,Y -628.738,Z 308.372,A 0.000,B 0.000,C 90.000,E1 282.883} C_DIS
LIN {X 0.090,Y -624.504,Z 308.356,A 0.000,B 0.000,C 90.000,E1 280.074} C_DIS
LIN {X 0.262,Y -621.831,Z 308.343,A 0.000,B 0.000,C 90.000,E1 277.757} C_DIS
LIN {X 0.215,Y -619.871,Z 308.330,A 0.000,B 0.000,C 90.000,E1 275.454} C_DIS
LIN {X -0.243,Y -619.018,Z 308.322,A 0.000,B 0.000,C 90.000,E1 273.955} C_DIS
LIN {X 0.153,Y -618.273,Z 308.309,A 0.000,B 0.000,C 90.000,E1 271.604} C_DIS
LIN {X 0.200,Y -618.153,Z 308.295,A 0.000,B 0.000,C 90.000,E1 269.026} C_DIS
LIN {X 0.251,Y -618.807,Z 308.283,A 0.000,B 0.000,C 90.000,E1 266.963} C_DIS
LIN {X -0.226,Y -619.951,Z 308.272,A 0.000,B 0.000,C 90.000,E1 264.951} C_DIS
LIN {X 0.022,Y -621.638,Z 308.260,A 0.000,B 0.000,C 90.000,E1 262.875} C_DIS
LIN {X 0.252,Y -624.664,Z 308.245,A 0.000,B 0.000,C 90.000,E1 260.038} C_DIS
LIN {X 0.304,Y -627.405,Z 308.233,A 0.000,B 0.000,C 90.000,E1 257.993} C_DIS
LIN {X 0.148,Y -630.026,Z 308.224,A 0.000,B 0.000,C 90.000,E1 256.228} C_DIS
LIN {X 0.227,Y -632.199,Z 308.215,A 0.000,B 0.000,C 90.000,E1 254.700} C_DIS
LIN {X -0.163,Y -633.046,Z 308.211,A 0.000,B 0.000,C 90.000,E1 253.976} C_DIS
LIN {X -0.298,Y -634.164,Z 308.204,A 0.000,B 0.000,C 90.000,E1 252.725} C_DIS
LIN {X -0.056,Y -634.847,Z 308.200,A 0.000,B 0.000,C 90.000,E1 251.945} C_DIS
LIN {X 0.208,Y -635.429,Z 308.194,A 0.000,B 0.000,C 90.000,E1 250.913} C_DIS
LIN {X -0.113,Y -635.595,Z 308.189,A 0.000,B 0.000,C 90.000,E1 249.934} C_DIS
LIN {X 0.163,Y -635.511,Z 308.183,A 0.000,B 0.000,C 90.000,E1 248.901} C_DIS
LIN {X 0.037,Y -635.067,Z 308.179,A 0.000,B 0.000,C 90.000,E1 248.156} C_DIS
LIN {X -0.089,Y -634.441,Z 308.174,A 0.000,B 0.000,C 90.000,E1 247.411} C_DIS
LIN {X -0.222,Y -633.542,Z 308.170,A 0.000,B 0.000,C 90.000,E1 246.666} C_DIS
LIN {X 0.211,Y -632.407,Z 308.166,A 0.000,B 0.000,C 90.000,E1 245.869} C_DIS
LIN {X 0.312,Y -631.021,Z 308.162,A 0.000,B 0.000,C 90.000,E1 245.101} C_DIS
LIN {X 0.132,Y -629.378,Z 308.158,A 0.000,B 0.000,C 90.000,E1 244.357} C_DIS
LIN {X 0.205,Y -627.564,Z 308.153,A 0.000,B 0.000,C 90.000,E1 243.589} C_DIS
LIN {X -0.297,Y -625.512,Z 308.149,A 0.000,B 0.000,C 90.000,E1 242.871} C_DIS
LIN {X 0.046,Y -621.845,Z 308.142,A 0.000,B 0.000,C 90.000,E1 241.563} C_DIS
LIN {X -0.239,Y -616.477,Z 308.132,A 0.000,B 0.000,C 90.000,E1 239.793} C_DIS
LIN {X 0.256,Y -612.559,Z 308.125,A 0.000,B 0.000,C 90.000,E1 238.456} C_DIS
LIN {X 0.160,Y -608.523,Z 308.118,A 0.000,B 0.000,C 90.000,E1 237.168} C_DIS
LIN {X 0.253,Y -603.818,Z 308.109,A 0.000,B 0.000,C 90.000,E1 235.595} C_DIS
LIN {X 0.093,Y -598.939,Z 308.100,A 0.000,B 0.000,C 90.000,E1 234.036} C_DIS
LIN {X 0.084,Y -594.493,Z 308.093,A 0.000,B 0.000,C 90.000,E1 232.718} C_DIS
LIN {X 0.079,Y -589.122,Z 308.084,A 0.000,B 0.000,C 90.000,E1 231.126} C_DIS
LIN {X -0.304,Y -584.757,Z 308.077,A 0.000,B 0.000,C 90.000,E1 229.828} C_DIS
LIN {X -0.157,Y -577.011,Z 308.063,A 0.000,B 0.000,C 90.000,E1 227.391} C_DIS
LIN {X -0.340,Y -572.815,Z 308.056,A 0.000,B 0.000,C 90.000,E1 226.053} C_DIS
LIN {X -0.002,Y -566.827,Z 308.045,A 0.000,B 0.000,C 90.000,E1 224.109} C_DIS
LIN {X 0.113,Y -561.838,Z 308.036,A 0.000,B 0.000,C 90.000,E1 222.447} C_DIS
LIN {X 0.081,Y -557.662,Z 308.028,A 0.000,B 0.000,C 90.000,E1 221.067} C_DIS
LIN {X -0.031,Y -553.445,Z 308.021,A 0.000,B 0.000,C 90.000,E1 219.688} C_DIS
LIN {X -0.091,Y -548.403,Z 308.011,A 0.000,B 0.000,C 90.000,E1 218.016} C_DIS
LIN {X 0.143,Y -544.160,Z 308.003,A 0.000,B 0.000,C 90.000,E1 216.583} C_DIS
LIN {X 0.046,Y -536.854,Z 307.989,A 0.000,B 0.000,C 90.000,E1 214.040} C_DIS
LIN {X 0.206,Y -534.518,Z 307.984,A 0.000,B 0.000,C 90.000,E1 213.166} C_DIS
LIN {X -0.020,Y -529.052,Z 307.973,A 0.000,B 0.000,C 90.000,E1 211.180} C_DIS
LIN {X -0.161,Y -524.700,Z 307.964,A 0.000,B 0.000,C 90.000,E1 209.461} C_DIS
LIN {X 0.194,Y -519.618,Z 307.952,A 0.000,B 0.000,C 90.000,E1 207.385} C_DIS
LIN {X 0.167,Y -516.099,Z 307.944,A 0.000,B 0.000,C 90.000,E1 205.924} C_DIS
LIN {X -0.266,Y -512.133,Z 307.934,A 0.000,B 0.000,C 90.000,E1 204.207} C_DIS
LIN {X 0.047,Y -507.550,Z 307.923,A 0.000,B 0.000,C 90.000,E1 202.099} C_DIS
LIN {X 0.232,Y -503.270,Z 307.911,A 0.000,B 0.000,C 90.000,E1 199.993} C_DIS
LIN {X -0.210,Y -499.100,Z 307.900,A 0.000,B 0.000,C 90.000,E1 197.946} C_DIS
LIN {X 0.201,Y -495.173,Z 307.888,A 0.000,B 0.000,C 90.000,E1 195.788} C_DIS
LIN {X 0.152,Y -490.725,Z 307.873,A 0.000,B 0.000,C 90.000,E1 193.063} C_DIS
LIN {X 0.192,Y -488.313,Z 307.864,A 0.000,B 0.000,C 90.000,E1 191.535} C_DIS
LIN {X -0.020,Y -484.281,Z 307.849,A 0.000,B 0.000,C 90.000,E1 188.803} C_DIS
LIN {X -0.146,Y -481.375,Z 307.837,A 0.000,B 0.000,C 90.000,E1 186.663} C_DIS
LIN {X -0.045,Y -479.466,Z 307.828,A 0.000,B 0.000,C 90.000,E1 185.106} C_DIS
LIN {X 0.073,Y -477.044,Z 307.816,A 0.000,B 0.000,C 90.000,E1 182.922} C_DIS
LIN {X 0.017,Y -475.431,Z 307.808,A 0.000,B 0.000,C 90.000,E1 181.375} C_DIS
LIN {X 0.076,Y -472.842,Z 307.789,A 0.000,B 0.000,C 90.000,E1 177.936} C_DIS
LIN {X -0.170,Y -471.375,Z 307.771,A 0.000,B 0.000,C 90.000,E1 174.837} C_DIS
LIN {X 0.075,Y -470.754,Z 307.757,A 0.000,B 0.000,C 90.000,E1 172.299} C_DIS
LIN {X 0.077,Y -470.609,Z 307.740,A 0.000,B 0.000,C 90.000,E1 169.162} C_DIS
LIN {X -0.059,Y -471.548,Z 307.717,A 0.000,B 0.000,C 90.000,E1 165.102} C_DIS
LIN {X -0.252,Y -473.019,Z 307.702,A 0.000,B 0.000,C 90.000,E1 162.308} C_DIS
LIN {X 0.215,Y -474.770,Z 307.688,A 0.000,B 0.000,C 90.000,E1 159.752} C_DIS
LIN {X -0.133,Y -476.586,Z 307.676,A 0.000,B 0.000,C 90.000,E1 157.614} C_DIS
LIN {X 0.119,Y -479.066,Z 307.664,A 0.000,B 0.000,C 90.000,E1 155.409} C_DIS
LIN {X -0.015,Y -483.808,Z 307.645,A 0.000,B 0.000,C 90.000,E1 152.025} C_DIS
LIN {X -0.116,Y -489.782,Z 307.626,A 0.000,B 0.000,C 90.000,E1 148.663} C_DIS
LIN {X 0.149,Y -494.100,Z 307.614,A 0.000,B 0.000,C 90.000,E1 146.501} C_DIS
LIN {X -0.024,Y -498.537,Z 307.602,A 0.000,B 0.000,C 90.000,E1 144.402} C_DIS
LIN {X -0.131,Y -500.976,Z 307.596,A 0.000,B 0.000,C 90.000,E1 143.210} C_DIS
LIN {X -0.021,Y -503.897,Z 307.587,A 0.000,B 0.000,C 90.000,E1 141.698} C_DIS
LIN {X -0.148,Y -505.988,Z 307.581,A 0.000,B 0.000,C 90.000,E1 140.517} C_DIS
LIN {X -0.143,Y -507.393,Z 307.576,A 0.000,B 0.000,C 90.000,E1 139.622} C_DIS
LIN {X 0.109,Y -508.986,Z 307.569,A 0.000,B 0.000,C 90.000,E1 138.405} C_DIS
LIN {X -0.237,Y -509.965,Z 307.564,A 0.000,B 0.000,C 90.000,E1 137.553} C_DIS
LIN {X 0.150,Y -510.669,Z 307.559,A 0.000,B 0.000,C 90.000,E1 136.620} C_DIS
LIN {X 0.174,Y -511.172,Z 307.554,A 0.000,B 0.000,C 90.000,E1 135.729} C_DIS
LIN {X 0.208,Y -511.360,Z 307.549,A 0.000,B 0.000,C 90.000,E1 134.838} C_DIS
LIN {X 0.242,Y -511.309,Z 307.544,A 0.000,B 0.000,C 90.000,E1 133.947} C_DIS
LIN {X -0.078,Y -510.996,Z 307.539,A 0.000,B 0.000,C 90.000,E1 133.095} C_DIS
LIN {X -0.151,Y -510.127,Z 307.533,A 0.000,B 0.000,C 90.000,E1 131.919} C_DIS
LIN {X 0.237,Y -509.229,Z 307.528,A 0.000,B 0.000,C 90.000,E1 130.987} C_DIS
LIN {X 0.085,Y -507.463,Z 307.520,A 0.000,B 0.000,C 90.000,E1 129.519} C_DIS
LIN {X 0.118,Y -504.974,Z 307.510,A 0.000,B 0.000,C 90.000,E1 127.729} C_DIS
LIN {X -0.307,Y -503.232,Z 307.503,A 0.000,B 0.000,C 90.000,E1 126.583} C_DIS
LIN {X -0.059,Y -501.287,Z 307.496,A 0.000,B 0.000,C 90.000,E1 125.358} C_DIS
LIN {X 0.275,Y -499.149,Z 307.490,A 0.000,B 0.000,C 90.000,E1 124.119} C_DIS
LIN {X 0.025,Y -497.458,Z 307.485,A 0.000,B 0.000,C 90.000,E1 123.245} C_DIS
LIN {X -0.254,Y -493.921,Z 307.475,A 0.000,B 0.000,C 90.000,E1 121.465} C_DIS
LIN {X -0.202,Y -489.629,Z 307.463,A 0.000,B 0.000,C 90.000,E1 119.333} C_DIS
LIN {X 0.112,Y -486.580,Z 307.454,A 0.000,B 0.000,C 90.000,E1 117.769} C_DIS
LIN {X 0.143,Y -483.482,Z 307.446,A 0.000,B 0.000,C 90.000,E1 116.232} C_DIS
LIN {X 0.103,Y -479.777,Z 307.436,A 0.000,B 0.000,C 90.000,E1 114.387} C_DIS
LIN {X 0.194,Y -475.483,Z 307.424,A 0.000,B 0.000,C 90.000,E1 112.206} C_DIS
LIN {X 0.090,Y -473.067,Z 307.417,A 0.000,B 0.000,C 90.000,E1 110.972} C_DIS
LIN {X 0.189,Y -470.089,Z 307.408,A 0.000,B 0.000,C 90.000,E1 109.396} C_DIS
LIN {X -0.131,Y -464.381,Z 307.391,A 0.000,B 0.000,C 90.000,E1 106.315} C_DIS
LIN {X -0.172,Y -464.392,Z 307.391,A 0.000,B 0.000,C 90.000,E1 106.315} C_DIS
LIN {X -0.040,Y -467.514,Z 307.383,A 0.000,B 0.000,C 90.000,E1 105.009} C_DIS
LIN {X -0.235,Y -468.097,Z 307.382,A 0.000,B 0.000,C 90.000,E1 104.717} C_DIS
LIN {X -0.096,Y -475.756,Z 307.357,A 0.000,B 0.000,C 90.000,E1 100.310} C_DIS
LIN {X 0.209,Y -476.285,Z 307.356,A 0.000,B 0.000,C 90.000,E1 99.962} C_DIS
LIN {X 0.158,Y -481.755,Z 307.331,A 0.000,B 0.000,C 90.000,E1 95.625} C_DIS
LIN {X 0.005,Y -482.163,Z 307.330,A 0.000,B 0.000,C 90.000,E1 95.334} C_DIS
LIN {X -0.066,Y -485.285,Z 307.306,A 0.000,B 0.000,C 90.000,E1 91.031} C_DIS
LIN {X -0.241,Y -485.538,Z 307.304,A 0.000,B 0.000,C 90.000,E1 90.745} C_DIS
LIN {X -0.034,Y -486.309,Z 307.282,A 0.000,B 0.000,C 90.000,E1 86.731} C_DIS
LIN {X 0.101,Y -486.319,Z 307.278,A 0.000,B 0.000,C 90.000,E1 86.102} C_DIS
LIN {X 0.173,Y -484.623,Z 307.253,A 0.000,B 0.000,C 90.000,E1 81.489} C_DIS
LIN {X 0.054,Y -480.552,Z 307.227,A 0.000,B 0.000,C 90.000,E1 76.881} C_DIS
LIN {X -0.143,Y -475.592,Z 307.208,A 0.000,B 0.000,C 90.000,E1 73.378} C_DIS
LIN {X 0.215,Y -481.355,Z 307.194,A 0.000,B 0.000,C 90.000,E1 70.967} C_DIS
LIN {X -0.063,Y -488.645,Z 307.179,A 0.000,B 0.000,C 90.000,E1 68.230} C_DIS
LIN {X -0.104,Y -494.554,Z 307.167,A 0.000,B 0.000,C 90.000,E1 66.102} C_DIS
LIN {X -0.102,Y -498.774,Z 307.159,A 0.000,B 0.000,C 90.000,E1 64.588} C_DIS
LIN {X 0.266,Y -503.960,Z 307.149,A 0.000,B 0.000,C 90.000,E1 62.743} C_DIS
LIN {X 0.134,Y -507.418,Z 307.142,A 0.000,B 0.000,C 90.000,E1 61.563} C_DIS
LIN {X 0.139,Y -511.761,Z 307.134,A 0.000,B 0.000,C 90.000,E1 60.078} C_DIS
LIN {X 0.026,Y -516.105,Z 307.126,A 0.000,B 0.000,C 90.000,E1 58.614} C_DIS
LIN {X -0.110,Y -519.537,Z 307.119,A 0.000,B 0.000,C 90.000,E1 57.454} C_DIS
LIN {X 0.145,Y -524.633,Z 307.109,A 0.000,B 0.000,C 90.000,E1 55.674} C_DIS
LIN {X -0.025,Y -528.632,Z 307.101,A 0.000,B 0.000,C 90.000,E1 54.242} C_DIS
LIN {X 0.313,Y -532.346,Z 307.093,A 0.000,B 0.000,C 90.000,E1 52.763} C_DIS
LIN {X -0.135,Y -535.664,Z 307.085,A 0.000,B 0.000,C 90.000,E1 51.376} C_DIS
LIN {X -0.131,Y -537.480,Z 307.081,A 0.000,B 0.000,C 90.000,E1 50.517} C_DIS
LIN {X -0.168,Y -539.734,Z 307.074,A 0.000,B 0.000,C 90.000,E1 49.380} C_DIS
LIN {X 0.217,Y -542.634,Z 307.065,A 0.000,B 0.000,C 90.000,E1 47.634} C_DIS
LIN {X 0.215,Y -543.533,Z 307.062,A 0.000,B 0.000,C 90.000,E1 47.067} C_DIS
LIN {X -0.121,Y -545.629,Z 307.052,A 0.000,B 0.000,C 90.000,E1 45.405} C_DIS
LIN {X -0.068,Y -546.517,Z 307.046,A 0.000,B 0.000,C 90.000,E1 44.271} C_DIS
LIN {X -0.007,Y -547.264,Z 307.040,A 0.000,B 0.000,C 90.000,E1 43.137} C_DIS
LIN {X 0.055,Y -547.699,Z 307.035,A 0.000,B 0.000,C 90.000,E1 42.285} C_DIS
LIN {X 0.161,Y -548.019,Z 307.029,A 0.000,B 0.000,C 90.000,E1 41.148} C_DIS
LIN {X -0.124,Y -548.166,Z 307.024,A 0.000,B 0.000,C 90.000,E1 40.334} C_DIS
LIN {X -0.056,Y -548.143,Z 307.019,A 0.000,B 0.000,C 90.000,E1 39.483} C_DIS
LIN {X 0.086,Y -547.924,Z 307.015,A 0.000,B 0.000,C 90.000,E1 38.624} C_DIS
LIN {X -0.200,Y -547.499,Z 307.010,A 0.000,B 0.000,C 90.000,E1 37.810} C_DIS
LIN {X -0.011,Y -546.744,Z 307.004,A 0.000,B 0.000,C 90.000,E1 36.664} C_DIS
LIN {X 0.163,Y -545.849,Z 306.997,A 0.000,B 0.000,C 90.000,E1 35.518} C_DIS
LIN {X 0.074,Y -544.342,Z 306.988,A 0.000,B 0.000,C 90.000,E1 33.833} C_DIS
LIN {X 0.077,Y -542.984,Z 306.980,A 0.000,B 0.000,C 90.000,E1 32.418} C_DIS
LIN {X 0.280,Y -540.878,Z 306.968,A 0.000,B 0.000,C 90.000,E1 30.129} C_DIS
LIN {X 0.141,Y -539.036,Z 306.957,A 0.000,B 0.000,C 90.000,E1 28.153} C_DIS
LIN {X -0.276,Y -537.414,Z 306.947,A 0.000,B 0.000,C 90.000,E1 26.488} C_DIS
LIN {X 0.175,Y -535.257,Z 306.934,A 0.000,B 0.000,C 90.000,E1 24.155} C_DIS
LIN {X 0.055,Y -533.130,Z 306.920,A 0.000,B 0.000,C 90.000,E1 21.589} C_DIS
LIN {X -0.227,Y -531.342,Z 306.906,A 0.000,B 0.000,C 90.000,E1 19.033} C_DIS
LIN {X 0.080,Y -530.143,Z 306.894,A 0.000,B 0.000,C 90.000,E1 16.985} C_DIS
LIN {X 0.002,Y -529.518,Z 306.886,A 0.000,B 0.000,C 90.000,E1 15.552} C_DIS
LIN {X 0.143,Y -528.619,Z 306.872,A 0.000,B 0.000,C 90.000,E1 12.939} C_DIS
LIN {X -0.226,Y -528.343,Z 306.864,A 0.000,B 0.000,C 90.000,E1 11.535} C_DIS
LIN {X -0.146,Y -528.126,Z 306.854,A 0.000,B 0.000,C 90.000,E1 9.792} C_DIS
LIN {X -0.037,Y -528.127,Z 306.848,A 0.000,B 0.000,C 90.000,E1 8.624} C_DIS
LIN {X -0.099,Y -528.484,Z 306.833,A 0.000,B 0.000,C 90.000,E1 6.030} C_DIS
LIN {X -0.137,Y -529.056,Z 306.822,A 0.000,B 0.000,C 90.000,E1 4.012} C_DIS
LIN {X -0.269,Y -529.967,Z 306.811,A 0.000,B 0.000,C 90.000,E1 2.007} C_DIS
LIN {X 0.000,Y -530.965,Z 306.800,A 0.000,B 0.000,C 90.000,E1 360.000} C_DIS
LIN {X 0.123,Y -532.916,Z 306.786,A 0.000,B 0.000,C 90.000,E1 357.478} C_DIS
LIN {X 0.123,Y -534.747,Z 306.775,A 0.000,B 0.000,C 90.000,E1 355.469} C_DIS
LIN {X 0.203,Y -536.842,Z 306.764,A 0.000,B 0.000,C 90.000,E1 353.457} C_DIS
LIN {X 0.093,Y -545.060,Z 306.737,A 0.000,B 0.000,C 90.000,E1 348.634} C_DIS
LIN {X 0.026,Y -551.918,Z 306.721,A 0.000,B 0.000,C 90.000,E1 345.825} C_DIS
LIN {X -0.196,Y -557.910,Z 306.709,A 0.000,B 0.000,C 90.000,E1 343.614} C_DIS
LIN {X -0.241,Y -564.175,Z 306.697,A 0.000,B 0.000,C 90.000,E1 341.402} C_DIS
LIN {X -0.250,Y -569.067,Z 306.687,A 0.000,B 0.000,C 90.000,E1 339.752} C_DIS
LIN {X 0.049,Y -575.983,Z 306.675,A 0.000,B 0.000,C 90.000,E1 337.539} C_DIS
LIN {X -0.265,Y -579.573,Z 306.669,A 0.000,B 0.000,C 90.000,E1 336.485} C_DIS
LIN {X 0.233,Y -583.198,Z 306.663,A 0.000,B 0.000,C 90.000,E1 335.357} C_DIS
LIN {X -0.093,Y -589.901,Z 306.653,A 0.000,B 0.000,C 90.000,E1 333.512} C_DIS
LIN {X 0.191,Y -594.635,Z 306.645,A 0.000,B 0.000,C 90.000,E1 332.153} C_DIS
LIN {X 0.036,Y -599.185,Z 306.638,A 0.000,B 0.000,C 90.000,E1 330.845} C_DIS
LIN {X 0.125,Y -605.622,Z 306.628,A 0.000,B 0.000,C 90.000,E1 328.997} C_DIS
LIN {X 0.161,Y -612.013,Z 306.618,A 0.000,B 0.000,C 90.000,E1 327.168} C_DIS
LIN {X -0.171,Y -618.351,Z 306.608,A 0.000,B 0.000,C 90.000,E1 325.388} C_DIS
LIN {X -0.130,Y -621.934,Z 306.602,A 0.000,B 0.000,C 90.000,E1 324.356} C_DIS
LIN {X 0.156,Y -626.052,Z 306.595,A 0.000,B 0.000,C 90.000,E1 323.050} C_DIS
LIN {X 0.172,Y -629.126,Z 306.589,A 0.000,B 0.000,C 90.000,E1 322.029} C_DIS
LIN {X -0.051,Y -634.325,Z 306.579,A 0.000,B 0.000,C 90.000,E1 320.275} C_DIS
LIN {X -0.141,Y -638.809,Z 306.571,A 0.000,B 0.000,C 90.000,E1 318.771} C_DIS
LIN {X 0.362,Y -642.340,Z 306.564,A 0.000,B 0.000,C 90.000,E1 317.472} C_DIS
LIN {X 0.253,Y -648.204,Z 306.553,A 0.000,B 0.000,C 90.000,E1 315.486} C_DIS
LIN {X -0.026,Y -651.941,Z 306.546,A 0.000,B 0.000,C 90.000,E1 314.271} C_DIS
LIN {X 0.223,Y -655.338,Z 306.539,A 0.000,B 0.000,C 90.000,E1 313.014} C_DIS
LIN {X -0.400,Y -658.580,Z 306.532,A 0.000,B 0.000,C 90.000,E1 311.838} C_DIS
LIN {X 0.446,Y -661.558,Z 306.525,A 0.000,B 0.000,C 90.000,E1 310.539} C_DIS
LIN {X 0.427,Y -663.656,Z 306.520,A 0.000,B 0.000,C 90.000,E1 309.564} C_DIS
LIN {X -0.007,Y -666.128,Z 306.513,A 0.000,B 0.000,C 90.000,E1 308.382} C_DIS
LIN {X -0.388,Y -667.866,Z 306.508,A 0.000,B 0.000,C 90.000,E1 307.443} C_DIS
LIN {X 0.210,Y -668.974,Z 306.504,A 0.000,B 0.000,C 90.000,E1 306.664} C_DIS
LIN {X -0.138,Y -670.260,Z 306.498,A 0.000,B 0.000,C 90.000,E1 305.724} C_DIS
LIN {X 0.069,Y -671.023,Z 306.493,A 0.000,B 0.000,C 90.000,E1 304.739} C_DIS
LIN {X 0.317,Y -671.320,Z 306.489,A 0.000,B 0.000,C 90.000,E1 303.992} C_DIS
LIN {X 0.014,Y -671.403,Z 306.485,A 0.000,B 0.000,C 90.000,E1 303.293} C_DIS
LIN {X -0.142,Y -671.235,Z 306.480,A 0.000,B 0.000,C 90.000,E1 302.339} C_DIS
LIN {X 0.112,Y -670.751,Z 306.476,A 0.000,B 0.000,C 90.000,E1 301.592} C_DIS
LIN {X -0.402,Y -669.547,Z 306.470,A 0.000,B 0.000,C 90.000,E1 300.669} C_DIS
LIN {X -0.014,Y -667.804,Z 306.465,A 0.000,B 0.000,C 90.000,E1 299.667} C_DIS
LIN {X -0.133,Y -666.242,Z 306.461,A 0.000,B 0.000,C 90.000,E1 298.949} C_DIS
LIN {X -0.116,Y -664.053,Z 306.455,A 0.000,B 0.000,C 90.000,E1 297.975} C_DIS
LIN {X 0.009,Y -661.063,Z 306.449,A 0.000,B 0.000,C 90.000,E1 296.744} C_DIS
LIN {X -0.209,Y -657.971,Z 306.442,A 0.000,B 0.000,C 90.000,E1 295.540} C_DIS
LIN {X 0.235,Y -653.998,Z 306.434,A 0.000,B 0.000,C 90.000,E1 294.027} C_DIS
LIN {X -0.085,Y -648.551,Z 306.423,A 0.000,B 0.000,C 90.000,E1 292.078} C_DIS
LIN {X -0.176,Y -645.280,Z 306.416,A 0.000,B 0.000,C 90.000,E1 290.844} C_DIS
LIN {X -0.223,Y -640.152,Z 306.405,A 0.000,B 0.000,C 90.000,E1 288.852} C_DIS
LIN {X 0.044,Y -634.235,Z 306.391,A 0.000,B 0.000,C 90.000,E1 286.315} C_DIS
LIN {X -0.003,Y -628.631,Z 306.375,A 0.000,B 0.000,C 90.000,E1 283.536} C_DIS
LIN {X -0.111,Y -623.734,Z 306.358,A 0.000,B 0.000,C 90.000,E1 280.489} C_DIS
LIN {X 0.084,Y -621.520,Z 306.348,A 0.000,B 0.000,C 90.000,E1 278.681} C_DIS
LIN {X -0.230,Y -619.088,Z 306.334,A 0.000,B 0.000,C 90.000,E1 276.144} C_DIS
LIN {X -0.088,Y -617.815,Z 306.323,A 0.000,B 0.000,C 90.000,E1 274.073} C_DIS
LIN {X 0.002,Y -616.913,Z 306.305,A 0.000,B 0.000,C 90.000,E1 270.974} C_DIS
LIN {X 0.025,Y -617.191,Z 306.288,A 0.000,B 0.000,C 90.000,E1 267.879} C_DIS
LIN {X 0.085,Y -618.477,Z 306.274,A 0.000,B 0.000,C 90.000,E1 265.298} C_DIS
LIN {X -0.037,Y -620.320,Z 306.261,A 0.000,B 0.000,C 90.000,E1 262.996} C_DIS
LIN {X -0.098,Y -623.683,Z 306.244,A 0.000,B 0.000,C 90.000,E1 259.926} C_DIS
LIN {X -0.082,Y -626.451,Z 306.233,A 0.000,B 0.000,C 90.000,E1 257.881} C_DIS
LIN {X -0.073,Y -628.746,Z 306.224,A 0.000,B 0.000,C 90.000,E1 256.353} C_DIS
LIN {X 0.138,Y -630.953,Z 306.216,A 0.000,B 0.000,C 90.000,E1 254.810} C_DIS
LIN {X -0.243,Y -631.602,Z 306.213,A 0.000,B 0.000,C 90.000,E1 254.338} C_DIS
LIN {X 0.200,Y -632.765,Z 306.206,A 0.000,B 0.000,C 90.000,E1 253.032} C_DIS
LIN {X -0.172,Y -633.697,Z 306.200,A 0.000,B 0.000,C 90.000,E1 252.054} C_DIS
LIN {X -0.123,Y -634.272,Z 306.195,A 0.000,B 0.000,C 90.000,E1 251.040} C_DIS
LIN {X 0.325,Y -634.497,Z 306.190,A 0.000,B 0.000,C 90.000,E1 250.242} C_DIS
LIN {X -0.205,Y -634.502,Z 306.183,A 0.000,B 0.000,C 90.000,E1 249.028} C_DIS
LIN {X 0.280,Y -633.947,Z 306.178,A 0.000,B 0.000,C 90.000,E1 247.975} C_DIS
LIN {X 0.140,Y -633.293,Z 306.174,A 0.000,B 0.000,C 90.000,E1 247.230} C_DIS
LIN {X -0.006,Y -632.370,Z 306.169,A 0.000,B 0.000,C 90.000,E1 246.485} C_DIS
LIN {X -0.165,Y -631.199,Z 306.165,A 0.000,B 0.000,C 90.000,E1 245.741} C_DIS
LIN {X -0.104,Y -630.327,Z 306.162,A 0.000,B 0.000,C 90.000,E1 245.229} C_DIS
LIN {X 0.009,Y -628.149,Z 306.157,A 0.000,B 0.000,C 90.000,E1 244.204} C_DIS
LIN {X 0.077,Y -626.300,Z 306.152,A 0.000,B 0.000,C 90.000,E1 243.435} C_DIS
LIN {X 0.127,Y -624.225,Z 306.148,A 0.000,B 0.000,C 90.000,E1 242.666} C_DIS
LIN {X 0.153,Y -620.555,Z 306.141,A 0.000,B 0.000,C 90.000,E1 241.385} C_DIS
LIN {X -0.151,Y -615.989,Z 306.133,A 0.000,B 0.000,C 90.000,E1 239.871} C_DIS
LIN {X 0.330,Y -612.067,Z 306.125,A 0.000,B 0.000,C 90.000,E1 238.535} C_DIS
LIN {X 0.221,Y -608.051,Z 306.118,A 0.000,B 0.000,C 90.000,E1 237.248} C_DIS
LIN {X -0.199,Y -603.334,Z 306.109,A 0.000,B 0.000,C 90.000,E1 235.722} C_DIS
LIN {X 0.126,Y -598.465,Z 306.101,A 0.000,B 0.000,C 90.000,E1 234.116} C_DIS
LIN {X -0.368,Y -594.023,Z 306.093,A 0.000,B 0.000,C 90.000,E1 232.844} C_DIS
LIN {X -0.002,Y -588.698,Z 306.085,A 0.000,B 0.000,C 90.000,E1 231.215} C_DIS
LIN {X -0.304,Y -584.348,Z 306.077,A 0.000,B 0.000,C 90.000,E1 229.908} C_DIS
LIN {X 0.107,Y -577.396,Z 306.065,A 0.000,B 0.000,C 90.000,E1 227.715} C_DIS
LIN {X 0.213,Y -574.101,Z 306.059,A 0.000,B 0.000,C 90.000,E1 226.620} C_DIS
LIN {X -0.139,Y -570.686,Z 306.053,A 0.000,B 0.000,C 90.000,E1 225.567} C_DIS
LIN {X -0.343,Y -565.589,Z 306.044,A 0.000,B 0.000,C 90.000,E1 223.947} C_DIS
LIN {X 0.074,Y -561.432,Z 306.036,A 0.000,B 0.000,C 90.000,E1 222.528} C_DIS
LIN {X 0.036,Y -557.272,Z 306.029,A 0.000,B 0.000,C 90.000,E1 221.148} C_DIS
LIN {X -0.080,Y -553.074,Z 306.021,A 0.000,B 0.000,C 90.000,E1 219.769} C_DIS
LIN {X -0.146,Y -547.990,Z 306.012,A 0.000,B 0.000,C 90.000,E1 218.096} C_DIS
LIN {X 0.082,Y -543.769,Z 306.004,A 0.000,B 0.000,C 90.000,E1 216.664} C_DIS
LIN {X -0.015,Y -535.638,Z 305.988,A 0.000,B 0.000,C 90.000,E1 213.833} C_DIS
LIN {X 0.236,Y -530.098,Z 305.977,A 0.000,B 0.000,C 90.000,E1 211.799} C_DIS
LIN {X -0.241,Y -524.174,Z 305.964,A 0.000,B 0.000,C 90.000,E1 209.539} C_DIS
LIN {X 0.109,Y -519.080,Z 305.953,A 0.000,B 0.000,C 90.000,E1 207.462} C_DIS
LIN {X -0.160,Y -515.556,Z 305.945,A 0.000,B 0.000,C 90.000,E1 206.027} C_DIS
LIN {X -0.148,Y -511.571,Z 305.935,A 0.000,B 0.000,C 90.000,E1 204.259} C_DIS
LIN {X -0.229,Y -506.400,Z 305.922,A 0.000,B 0.000,C 90.000,E1 201.897} C_DIS
LIN {X 0.216,Y -502.155,Z 305.910,A 0.000,B 0.000,C 90.000,E1 199.758} C_DIS
LIN {X -0.189,Y -497.514,Z 305.897,A 0.000,B 0.000,C 90.000,E1 197.402} C_DIS
LIN {X 0.173,Y -493.712,Z 305.885,A 0.000,B 0.000,C 90.000,E1 195.245} C_DIS
LIN {X 0.170,Y -490.373,Z 305.873,A 0.000,B 0.000,C 90.000,E1 193.119} C_DIS
LIN {X 0.200,Y -488.013,Z 305.865,A 0.000,B 0.000,C 90.000,E1 191.591} C_DIS
LIN {X 0.104,Y -484.477,Z 305.851,A 0.000,B 0.000,C 90.000,E1 189.151} C_DIS
LIN {X -0.159,Y -481.231,Z 305.837,A 0.000,B 0.000,C 90.000,E1 186.720} C_DIS
LIN {X -0.061,Y -479.351,Z 305.829,A 0.000,B 0.000,C 90.000,E1 185.163} C_DIS
LIN {X 0.053,Y -477.011,Z 305.817,A 0.000,B 0.000,C 90.000,E1 182.980} C_DIS
LIN {X -0.005,Y -475.455,Z 305.808,A 0.000,B 0.000,C 90.000,E1 181.432} C_DIS
LIN {X 0.056,Y -472.907,Z 305.789,A 0.000,B 0.000,C 90.000,E1 177.993} C_DIS
LIN {X -0.184,Y -471.460,Z 305.772,A 0.000,B 0.000,C 90.000,E1 174.894} C_DIS
LIN {X -0.221,Y -470.921,Z 305.759,A 0.000,B 0.000,C 90.000,E1 172.704} C_DIS
LIN {X -0.034,Y -470.645,Z 305.744,A 0.000,B 0.000,C 90.000,E1 169.859} C_DIS
LIN {X -0.099,Y -470.680,Z 305.738,A 0.000,B 0.000,C 90.000,E1 168.926} C_DIS
LIN {X -0.171,Y -471.558,Z 305.718,A 0.000,B 0.000,C 90.000,E1 165.172} C_DIS
LIN {X -0.053,Y -472.783,Z 305.704,A 0.000,B 0.000,C 90.000,E1 162.653} C_DIS
LIN {X 0.103,Y -474.533,Z 305.690,A 0.000,B 0.000,C 90.000,E1 160.134} C_DIS
LIN {X -0.106,Y -476.499,Z 305.676,A 0.000,B 0.000,C 90.000,E1 157.667} C_DIS
LIN {X -0.049,Y -478.856,Z 305.664,A 0.000,B 0.000,C 90.000,E1 155.485} C_DIS
LIN {X 0.230,Y -483.006,Z 305.647,A 0.000,B 0.000,C 90.000,E1 152.359} C_DIS
LIN {X 0.091,Y -488.765,Z 305.628,A 0.000,B 0.000,C 90.000,E1 148.997} C_DIS
LIN {X -0.094,Y -493.533,Z 305.614,A 0.000,B 0.000,C 90.000,E1 146.580} C_DIS
LIN {X -0.153,Y -497.236,Z 305.604,A 0.000,B 0.000,C 90.000,E1 144.769} C_DIS
LIN {X -0.111,Y -500.251,Z 305.596,A 0.000,B 0.000,C 90.000,E1 143.256} C_DIS
LIN {X -0.006,Y -503.085,Z 305.587,A 0.000,B 0.000,C 90.000,E1 141.743} C_DIS
LIN {X -0.139,Y -505.165,Z 305.581,A 0.000,B 0.000,C 90.000,E1 140.561} C_DIS
LIN {X -0.244,Y -507.012,Z 305.574,A 0.000,B 0.000,C 90.000,E1 139.380} C_DIS
LIN {X 0.004,Y -508.510,Z 305.568,A 0.000,B 0.000,C 90.000,E1 138.162} C_DIS
LIN {X 0.136,Y -509.146,Z 305.564,A 0.000,B 0.000,C 90.000,E1 137.553} C_DIS
LIN {X 0.035,Y -510.041,Z 305.558,A 0.000,B 0.000,C 90.000,E1 136.377} C_DIS
LIN {X -0.193,Y -510.372,Z 305.554,A 0.000,B 0.000,C 90.000,E1 135.810} C_DIS
LIN {X -0.170,Y -510.562,Z 305.549,A 0.000,B 0.000,C 90.000,E1 134.919} C_DIS
LIN {X -0.143,Y -510.527,Z 305.545,A 0.000,B 0.000,C 90.000,E1 134.028} C_DIS
LIN {X -0.224,Y -510.062,Z 305.538,A 0.000,B 0.000,C 90.000,E1 132.852} C_DIS
LIN {X 0.166,Y -509.390,Z 305.533,A 0.000,B 0.000,C 90.000,E1 131.919} C_DIS
LIN {X -0.173,Y -508.502,Z 305.528,A 0.000,B 0.000,C 90.000,E1 131.067} C_DIS
LIN {X -0.013,Y -506.733,Z 305.520,A 0.000,B 0.000,C 90.000,E1 129.564} C_DIS
LIN {X -0.313,Y -504.245,Z 305.510,A 0.000,B 0.000,C 90.000,E1 127.810} C_DIS
LIN {X -0.042,Y -502.493,Z 305.503,A 0.000,B 0.000,C 90.000,E1 126.583} C_DIS
LIN {X -0.097,Y -500.553,Z 305.497,A 0.000,B 0.000,C 90.000,E1 125.391} C_DIS
LIN {X -0.177,Y -498.409,Z 305.490,A 0.000,B 0.000,C 90.000,E1 124.199} C_DIS
LIN {X 0.118,Y -496.126,Z 305.483,A 0.000,B 0.000,C 90.000,E1 122.959} C_DIS
LIN {X -0.041,Y -493.187,Z 305.475,A 0.000,B 0.000,C 90.000,E1 121.465} C_DIS
LIN {X -0.010,Y -488.936,Z 305.463,A 0.000,B 0.000,C 90.000,E1 119.333} C_DIS
LIN {X 0.289,Y -485.880,Z 305.454,A 0.000,B 0.000,C 90.000,E1 117.769} C_DIS
LIN {X -0.127,Y -482.803,Z 305.446,A 0.000,B 0.000,C 90.000,E1 116.283} C_DIS
LIN {X 0.250,Y -479.115,Z 305.436,A 0.000,B 0.000,C 90.000,E1 114.387} C_DIS
LIN {X -0.118,Y -474.818,Z 305.424,A 0.000,B 0.000,C 90.000,E1 112.259} C_DIS
LIN {X 0.208,Y -472.427,Z 305.417,A 0.000,B 0.000,C 90.000,E1 110.972} C_DIS
LIN {X -0.149,Y -469.476,Z 305.408,A 0.000,B 0.000,C 90.000,E1 109.450} C_DIS
LIN {X -0.030,Y -464.072,Z 305.391,A 0.000,B 0.000,C 90.000,E1 106.441} C_DIS
LIN {X -0.070,Y -464.074,Z 305.391,A 0.000,B 0.000,C 90.000,E1 106.441} C_DIS
LIN {X 0.041,Y -467.489,Z 305.383,A 0.000,B 0.000,C 90.000,E1 105.009} C_DIS
LIN {X -0.154,Y -468.083,Z 305.382,A 0.000,B 0.000,C 90.000,E1 104.717} C_DIS
LIN {X -0.015,Y -475.736,Z 305.357,A 0.000,B 0.000,C 90.000,E1 100.310} C_DIS
LIN {X -0.178,Y -476.276,Z 305.356,A 0.000,B 0.000,C 90.000,E1 100.018} C_DIS
LIN {X -0.241,Y -481.739,Z 305.331,A 0.000,B 0.000,C 90.000,E1 95.682} C_DIS
LIN {X 0.087,Y -482.158,Z 305.330,A 0.000,B 0.000,C 90.000,E1 95.334} C_DIS
LIN {X -0.159,Y -485.538,Z 305.304,A 0.000,B 0.000,C 90.000,E1 90.745} C_DIS
LIN {X 0.048,Y -486.304,Z 305.282,A 0.000,B 0.000,C 90.000,E1 86.731} C_DIS
LIN {X 0.182,Y -486.327,Z 305.279,A 0.000,B 0.000,C 90.000,E1 86.102} C_DIS
LIN {X -0.224,Y -484.632,Z 305.253,A 0.000,B 0.000,C 90.000,E1 81.546} C_DIS
LIN {X 0.135,Y -480.559,Z 305.227,A 0.000,B 0.000,C 90.000,E1 76.881} C_DIS
LIN {X -0.172,Y -475.346,Z 305.207,A 0.000,B 0.000,C 90.000,E1 73.196} C_DIS
LIN {X -0.050,Y -481.397,Z 305.193,A 0.000,B 0.000,C 90.000,E1 70.678} C_DIS
LIN {X -0.036,Y -486.239,Z 305.182,A 0.000,B 0.000,C 90.000,E1 68.827} C_DIS
LIN {X 0.070,Y -490.435,Z 305.174,A 0.000,B 0.000,C 90.000,E1 67.283} C_DIS
LIN {X -0.162,Y -495.523,Z 305.164,A 0.000,B 0.000,C 90.000,E1 65.485} C_DIS
LIN {X -0.263,Y -501.490,Z 305.152,A 0.000,B 0.000,C 90.000,E1 63.384} C_DIS
LIN {X 0.082,Y -505.851,Z 305.144,A 0.000,B 0.000,C 90.000,E1 61.847} C_DIS
LIN {X -0.064,Y -511.029,Z 305.134,A 0.000,B 0.000,C 90.000,E1 60.078} C_DIS
LIN {X 0.164,Y -514.544,Z 305.127,A 0.000,B 0.000,C 90.000,E1 58.869} C_DIS
LIN {X 0.098,Y -518.822,Z 305.119,A 0.000,B 0.000,C 90.000,E1 57.406} C_DIS
LIN {X -0.103,Y -523.895,Z 305.109,A 0.000,B 0.000,C 90.000,E1 55.674} C_DIS
LIN {X 0.172,Y -527.146,Z 305.103,A 0.000,B 0.000,C 90.000,E1 54.482} C_DIS
LIN {X 0.051,Y -530.916,Z 305.095,A 0.000,B 0.000,C 90.000,E1 53.050} C_DIS
LIN {X -0.005,Y -534.297,Z 305.087,A 0.000,B 0.000,C 90.000,E1 51.618} C_DIS
LIN {X 0.323,Y -536.195,Z 305.082,A 0.000,B 0.000,C 90.000,E1 50.723} C_DIS
LIN {X 0.279,Y -539.022,Z 305.074,A 0.000,B 0.000,C 90.000,E1 49.299} C_DIS
LIN {X -0.124,Y -541.471,Z 305.066,A 0.000,B 0.000,C 90.000,E1 47.919} C_DIS
LIN {X -0.120,Y -542.804,Z 305.061,A 0.000,B 0.000,C 90.000,E1 47.067} C_DIS
LIN {X -0.095,Y -544.561,Z 305.054,A 0.000,B 0.000,C 90.000,E1 45.648} C_DIS
LIN {X -0.078,Y -545.105,Z 305.050,A 0.000,B 0.000,C 90.000,E1 45.081} C_DIS
LIN {X -0.033,Y -545.952,Z 305.044,A 0.000,B 0.000,C 90.000,E1 43.947} C_DIS
LIN {X 0.018,Y -546.473,Z 305.039,A 0.000,B 0.000,C 90.000,E1 43.095} C_DIS
LIN {X 0.070,Y -547.020,Z 305.033,A 0.000,B 0.000,C 90.000,E1 41.962} C_DIS
LIN {X 0.164,Y -547.296,Z 305.027,A 0.000,B 0.000,C 90.000,E1 40.825} C_DIS
LIN {X -0.089,Y -547.390,Z 305.021,A 0.000,B 0.000,C 90.000,E1 39.725} C_DIS
LIN {X -0.036,Y -547.256,Z 305.016,A 0.000,B 0.000,C 90.000,E1 38.874} C_DIS
LIN {X 0.140,Y -546.716,Z 305.010,A 0.000,B 0.000,C 90.000,E1 37.729} C_DIS
LIN {X 0.355,Y -545.770,Z 305.002,A 0.000,B 0.000,C 90.000,E1 36.297} C_DIS
LIN {X 0.234,Y -544.602,Z 304.994,A 0.000,B 0.000,C 90.000,E1 34.898} C_DIS
LIN {X 0.118,Y -543.108,Z 304.985,A 0.000,B 0.000,C 90.000,E1 33.214} C_DIS
LIN {X -0.170,Y -541.418,Z 304.975,A 0.000,B 0.000,C 90.000,E1 31.544} C_DIS
LIN {X -0.215,Y -540.123,Z 304.967,A 0.000,B 0.000,C 90.000,E1 30.129} C_DIS
LIN {X -0.087,Y -538.781,Z 304.959,A 0.000,B 0.000,C 90.000,E1 28.693} C_DIS
LIN {X 0.017,Y -537.427,Z 304.951,A 0.000,B 0.000,C 90.000,E1 27.257} C_DIS
LIN {X -0.154,Y -536.020,Z 304.944,A 0.000,B 0.000,C 90.000,E1 25.848} C_DIS
LIN {X -0.155,Y -534.423,Z 304.934,A 0.000,B 0.000,C 90.000,E1 24.131} C_DIS
LIN {X 0.071,Y -532.710,Z 304.923,A 0.000,B 0.000,C 90.000,E1 22.099} C_DIS
LIN {X 0.068,Y -531.573,Z 304.915,A 0.000,B 0.000,C 90.000,E1 20.663} C_DIS
LIN {X -0.136,Y -530.277,Z 304.904,A 0.000,B 0.000,C 90.000,E1 18.671} C_DIS
LIN {X -0.173,Y -528.830,Z 304.889,A 0.000,B 0.000,C 90.000,E1 16.079} C_DIS
LIN {X -0.209,Y -527.922,Z 304.876,A 0.000,B 0.000,C 90.000,E1 13.772} C_DIS
LIN {X 0.099,Y -527.439,Z 304.865,A 0.000,B 0.000,C 90.000,E1 11.715} C_DIS
LIN {X 0.279,Y -527.147,Z 304.854,A 0.000,B 0.000,C 90.000,E1 9.670} C_DIS
LIN {X -0.234,Y -527.127,Z 304.848,A 0.000,B 0.000,C 90.000,E1 8.568} C_DIS
LIN {X 0.254,Y -527.464,Z 304.833,A 0.000,B 0.000,C 90.000,E1 5.910} C_DIS
LIN {X 0.081,Y -528.267,Z 304.819,A 0.000,B 0.000,C 90.000,E1 3.326} C_DIS
LIN {X -0.022,Y -529.070,Z 304.809,A 0.000,B 0.000,C 90.000,E1 1.604} C_DIS
LIN {X 0.105,Y -531.580,Z 304.788,A 0.000,B 0.000,C 90.000,E1 357.764} C_DIS
LIN {X 0.063,Y -533.642,Z 304.775,A 0.000,B 0.000,C 90.000,E1 355.469} C_DIS
LIN {X 0.114,Y -535.730,Z 304.764,A 0.000,B 0.000,C 90.000,E1 353.457} C_DIS
LIN {X -0.066,Y -543.930,Z 304.737,A 0.000,B 0.000,C 90.000,E1 348.634} C_DIS
LIN {X -0.280,Y -550.027,Z 304.723,A 0.000,B 0.000,C 90.000,E1 346.117} C_DIS
LIN {X 0.101,Y -556.724,Z 304.709,A 0.000,B 0.000,C 90.000,E1 343.559} C_DIS
LIN {X -0.203,Y -563.766,Z 304.695,A 0.000,B 0.000,C 90.000,E1 341.094} C_DIS
LIN {X -0.074,Y -569.571,Z 304.684,A 0.000,B 0.000,C 90.000,E1 339.156} C_DIS
LIN {X -0.083,Y -576.657,Z 304.672,A 0.000,B 0.000,C 90.000,E1 336.975} C_DIS
LIN {X -0.144,Y -582.067,Z 304.663,A 0.000,B 0.000,C 90.000,E1 335.357} C_DIS
LIN {X 0.026,Y -588.767,Z 304.653,A 0.000,B 0.000,C 90.000,E1 333.461} C_DIS
LIN {X -0.240,Y -593.500,Z 304.645,A 0.000,B 0.000,C 90.000,E1 332.153} C_DIS
LIN {X 0.104,Y -598.049,Z 304.638,A 0.000,B 0.000,C 90.000,E1 330.795} C_DIS
LIN {X 0.156,Y -604.472,Z 304.628,A 0.000,B 0.000,C 90.000,E1 328.948} C_DIS
LIN {X 0.155,Y -610.841,Z 304.617,A 0.000,B 0.000,C 90.000,E1 327.120} C_DIS
LIN {X 0.136,Y -617.224,Z 304.607,A 0.000,B 0.000,C 90.000,E1 325.308} C_DIS
LIN {X 0.166,Y -620.858,Z 304.602,A 0.000,B 0.000,C 90.000,E1 324.276} C_DIS
LIN {X 0.063,Y -625.026,Z 304.595,A 0.000,B 0.000,C 90.000,E1 323.004} C_DIS
LIN {X 0.057,Y -628.114,Z 304.589,A 0.000,B 0.000,C 90.000,E1 321.984} C_DIS
LIN {X 0.204,Y -633.356,Z 304.579,A 0.000,B 0.000,C 90.000,E1 320.194} C_DIS
LIN {X 0.098,Y -637.857,Z 304.571,A 0.000,B 0.000,C 90.000,E1 318.690} C_DIS
LIN {X -0.232,Y -640.686,Z 304.565,A 0.000,B 0.000,C 90.000,E1 317.715} C_DIS
LIN {X -0.394,Y -646.492,Z 304.554,A 0.000,B 0.000,C 90.000,E1 315.729} C_DIS
LIN {X 0.216,Y -650.209,Z 304.547,A 0.000,B 0.000,C 90.000,E1 314.433} C_DIS
LIN {X 0.010,Y -652.998,Z 304.542,A 0.000,B 0.000,C 90.000,E1 313.461} C_DIS
LIN {X -0.170,Y -656.296,Z 304.535,A 0.000,B 0.000,C 90.000,E1 312.243} C_DIS
LIN {X 0.213,Y -658.184,Z 304.531,A 0.000,B 0.000,C 90.000,E1 311.472} C_DIS
LIN {X 0.126,Y -661.092,Z 304.524,A 0.000,B 0.000,C 90.000,E1 310.253} C_DIS
LIN {X 0.075,Y -663.641,Z 304.517,A 0.000,B 0.000,C 90.000,E1 309.036} C_DIS
LIN {X -0.338,Y -665.515,Z 304.512,A 0.000,B 0.000,C 90.000,E1 308.096} C_DIS
LIN {X 0.207,Y -667.207,Z 304.506,A 0.000,B 0.000,C 90.000,E1 307.076} C_DIS
LIN {X -0.165,Y -668.504,Z 304.501,A 0.000,B 0.000,C 90.000,E1 306.137} C_DIS
LIN {X -0.077,Y -669.123,Z 304.498,A 0.000,B 0.000,C 90.000,E1 305.644} C_DIS
LIN {X 0.147,Y -669.690,Z 304.494,A 0.000,B 0.000,C 90.000,E1 304.898} C_DIS
LIN {X 0.346,Y -670.060,Z 304.489,A 0.000,B 0.000,C 90.000,E1 303.913} C_DIS
LIN {X 0.175,Y -670.135,Z 304.483,A 0.000,B 0.000,C 90.000,E1 302.959} C_DIS
LIN {X -0.146,Y -669.910,Z 304.479,A 0.000,B 0.000,C 90.000,E1 302.260} C_DIS
LIN {X 0.158,Y -669.642,Z 304.477,A 0.000,B 0.000,C 90.000,E1 301.750} C_DIS
LIN {X -0.022,Y -668.457,Z 304.471,A 0.000,B 0.000,C 90.000,E1 300.797} C_DIS
LIN {X -0.289,Y -667.685,Z 304.468,A 0.000,B 0.000,C 90.000,E1 300.335} C_DIS
LIN {X 0.071,Y -665.819,Z 304.463,A 0.000,B 0.000,C 90.000,E1 299.333} C_DIS
LIN {X 0.221,Y -663.072,Z 304.456,A 0.000,B 0.000,C 90.000,E1 298.103} C_DIS
LIN {X 0.329,Y -660.090,Z 304.449,A 0.000,B 0.000,C 90.000,E1 296.873} C_DIS
LIN {X 0.216,Y -656.363,Z 304.441,A 0.000,B 0.000,C 90.000,E1 295.412} C_DIS
LIN {X 0.027,Y -652.377,Z 304.433,A 0.000,B 0.000,C 90.000,E1 293.951} C_DIS
LIN {X 0.012,Y -646.943,Z 304.422,A 0.000,B 0.000,C 90.000,E1 291.972} C_DIS
LIN {X -0.095,Y -643.653,Z 304.415,A 0.000,B 0.000,C 90.000,E1 290.737} C_DIS
LIN {X 0.338,Y -640.431,Z 304.408,A 0.000,B 0.000,C 90.000,E1 289.450} C_DIS
LIN {X -0.282,Y -636.716,Z 304.400,A 0.000,B 0.000,C 90.000,E1 288.000} C_DIS
LIN {X -0.135,Y -631.560,Z 304.387,A 0.000,B 0.000,C 90.000,E1 285.717} C_DIS
LIN {X 0.119,Y -627.122,Z 304.375,A 0.000,B 0.000,C 90.000,E1 283.411} C_DIS
LIN {X 0.214,Y -621.942,Z 304.356,A 0.000,B 0.000,C 90.000,E1 280.084} C_DIS
LIN {X -0.197,Y -619.276,Z 304.343,A 0.000,B 0.000,C 90.000,E1 277.814} C_DIS
LIN {X 0.069,Y -616.899,Z 304.326,A 0.000,B 0.000,C 90.000,E1 274.702} C_DIS
LIN {X -0.221,Y -615.752,Z 304.310,A 0.000,B 0.000,C 90.000,E1 271.892} C_DIS
LIN {X -0.226,Y -615.563,Z 304.302,A 0.000,B 0.000,C 90.000,E1 270.344} C_DIS
LIN {X -0.257,Y -616.179,Z 304.285,A 0.000,B 0.000,C 90.000,E1 267.249} C_DIS
LIN {X -0.162,Y -618.103,Z 304.267,A 0.000,B 0.000,C 90.000,E1 264.147} C_DIS
LIN {X -0.268,Y -619.687,Z 304.257,A 0.000,B 0.000,C 90.000,E1 262.356} C_DIS
LIN {X -0.180,Y -622.346,Z 304.245,A 0.000,B 0.000,C 90.000,E1 260.038} C_DIS
LIN {X -0.192,Y -625.135,Z 304.233,A 0.000,B 0.000,C 90.000,E1 257.993} C_DIS
LIN {X -0.202,Y -627.434,Z 304.225,A 0.000,B 0.000,C 90.000,E1 256.464} C_DIS
LIN {X -0.174,Y -629.671,Z 304.216,A 0.000,B 0.000,C 90.000,E1 254.936} C_DIS
LIN {X 0.017,Y -630.606,Z 304.212,A 0.000,B 0.000,C 90.000,E1 254.157} C_DIS
LIN {X 0.034,Y -631.567,Z 304.206,A 0.000,B 0.000,C 90.000,E1 253.142} C_DIS
LIN {X 0.063,Y -632.633,Z 304.199,A 0.000,B 0.000,C 90.000,E1 251.873} C_DIS
LIN {X 0.289,Y -633.095,Z 304.195,A 0.000,B 0.000,C 90.000,E1 251.094} C_DIS
LIN {X -0.061,Y -633.386,Z 304.190,A 0.000,B 0.000,C 90.000,E1 250.115} C_DIS
LIN {X 0.186,Y -633.391,Z 304.184,A 0.000,B 0.000,C 90.000,E1 249.082} C_DIS
LIN {X -0.165,Y -632.900,Z 304.178,A 0.000,B 0.000,C 90.000,E1 248.103} C_DIS
LIN {X 0.297,Y -632.010,Z 304.173,A 0.000,B 0.000,C 90.000,E1 247.050} C_DIS
LIN {X 0.135,Y -631.038,Z 304.168,A 0.000,B 0.000,C 90.000,E1 246.305} C_DIS
LIN {X 0.221,Y -629.819,Z 304.164,A 0.000,B 0.000,C 90.000,E1 245.537} C_DIS
LIN {X 0.035,Y -628.403,Z 304.160,A 0.000,B 0.000,C 90.000,E1 244.793} C_DIS
LIN {X 0.119,Y -626.178,Z 304.154,A 0.000,B 0.000,C 90.000,E1 243.768} C_DIS
LIN {X 0.162,Y -624.227,Z 304.150,A 0.000,B 0.000,C 90.000,E1 242.999} C_DIS
LIN {X 0.188,Y -621.374,Z 304.144,A 0.000,B 0.000,C 90.000,E1 241.975} C_DIS
LIN {X -0.087,Y -617.643,Z 304.137,A 0.000,B 0.000,C 90.000,E1 240.717} C_DIS
LIN {X 0.116,Y -613.825,Z 304.130,A 0.000,B 0.000,C 90.000,E1 239.410} C_DIS
LIN {X 0.037,Y -609.887,Z 304.123,A 0.000,B 0.000,C 90.000,E1 238.122} C_DIS
LIN {X 0.160,Y -605.110,Z 304.114,A 0.000,B 0.000,C 90.000,E1 236.548} C_DIS
LIN {X -0.069,Y -601.187,Z 304.107,A 0.000,B 0.000,C 90.000,E1 235.261} C_DIS
LIN {X 0.075,Y -597.901,Z 304.101,A 0.000,B 0.000,C 90.000,E1 234.196} C_DIS
LIN {X -0.072,Y -593.465,Z 304.094,A 0.000,B 0.000,C 90.000,E1 232.889} C_DIS
LIN {X 0.122,Y -587.322,Z 304.083,A 0.000,B 0.000,C 90.000,E1 231.009} C_DIS
LIN {X 0.168,Y -582.973,Z 304.076,A 0.000,B 0.000,C 90.000,E1 229.666} C_DIS
LIN {X 0.258,Y -575.320,Z 304.063,A 0.000,B 0.000,C 90.000,E1 227.229} C_DIS
LIN {X 0.044,Y -571.123,Z 304.055,A 0.000,B 0.000,C 90.000,E1 225.891} C_DIS
LIN {X -0.153,Y -566.004,Z 304.046,A 0.000,B 0.000,C 90.000,E1 224.271} C_DIS
LIN {X 0.273,Y -561.825,Z 304.038,A 0.000,B 0.000,C 90.000,E1 222.852} C_DIS
LIN {X -0.095,Y -556.853,Z 304.029,A 0.000,B 0.000,C 90.000,E1 221.229} C_DIS
LIN {X -0.151,Y -551.806,Z 304.020,A 0.000,B 0.000,C 90.000,E1 219.564} C_DIS
LIN {X -0.189,Y -545.846,Z 304.009,A 0.000,B 0.000,C 90.000,E1 217.604} C_DIS
LIN {X -0.028,Y -542.481,Z 304.003,A 0.000,B 0.000,C 90.000,E1 216.457} C_DIS
LIN {X -0.168,Y -535.152,Z 303.988,A 0.000,B 0.000,C 90.000,E1 213.913} C_DIS
LIN {X 0.077,Y -529.577,Z 303.977,A 0.000,B 0.000,C 90.000,E1 211.878} C_DIS
LIN {X -0.147,Y -523.606,Z 303.964,A 0.000,B 0.000,C 90.000,E1 209.589} C_DIS
LIN {X 0.177,Y -518.499,Z 303.953,A 0.000,B 0.000,C 90.000,E1 207.513} C_DIS
LIN {X 0.130,Y -514.967,Z 303.945,A 0.000,B 0.000,C 90.000,E1 206.052} C_DIS
LIN {X 0.140,Y -510.968,Z 303.935,A 0.000,B 0.000,C 90.000,E1 204.283} C_DIS
LIN {X 0.247,Y -505.846,Z 303.922,A 0.000,B 0.000,C 90.000,E1 201.897} C_DIS
LIN {X 0.200,Y -501.625,Z 303.910,A 0.000,B 0.000,C 90.000,E1 199.812} C_DIS
LIN {X -0.175,Y -496.506,Z 303.895,A 0.000,B 0.000,C 90.000,E1 197.149} C_DIS
LIN {X -0.064,Y -491.841,Z 303.880,A 0.000,B 0.000,C 90.000,E1 194.411} C_DIS
LIN {X -0.006,Y -489.521,Z 303.872,A 0.000,B 0.000,C 90.000,E1 192.883} C_DIS
LIN {X 0.154,Y -486.334,Z 303.860,A 0.000,B 0.000,C 90.000,E1 190.725} C_DIS
LIN {X 0.231,Y -483.398,Z 303.848,A 0.000,B 0.000,C 90.000,E1 188.568} C_DIS
LIN {X 0.222,Y -481.089,Z 303.838,A 0.000,B 0.000,C 90.000,E1 186.720} C_DIS
LIN {X -0.050,Y -478.543,Z 303.826,A 0.000,B 0.000,C 90.000,E1 184.588} C_DIS
LIN {X -0.051,Y -476.965,Z 303.817,A 0.000,B 0.000,C 90.000,E1 183.037} C_DIS
LIN {X -0.110,Y -475.457,Z 303.808,A 0.000,B 0.000,C 90.000,E1 181.489} C_DIS
LIN {X -0.049,Y -472.933,Z 303.789,A 0.000,B 0.000,C 90.000,E1 178.051} C_DIS
LIN {X -0.098,Y -471.635,Z 303.774,A 0.000,B 0.000,C 90.000,E1 175.241} C_DIS
LIN {X 0.148,Y -470.960,Z 303.760,A 0.000,B 0.000,C 90.000,E1 172.704} C_DIS
LIN {X 0.225,Y -470.666,Z 303.747,A 0.000,B 0.000,C 90.000,E1 170.500} C_DIS
LIN {X 0.271,Y -470.693,Z 303.739,A 0.000,B 0.000,C 90.000,E1 168.926} C_DIS
LIN {X 0.200,Y -471.533,Z 303.718,A 0.000,B 0.000,C 90.000,E1 165.172} C_DIS
LIN {X 0.177,Y -472.728,Z 303.704,A 0.000,B 0.000,C 90.000,E1 162.670} C_DIS
LIN {X 0.060,Y -474.246,Z 303.692,A 0.000,B 0.000,C 90.000,E1 160.496} C_DIS
LIN {X -0.155,Y -476.158,Z 303.678,A 0.000,B 0.000,C 90.000,E1 158.028} C_DIS
LIN {X -0.149,Y -479.368,Z 303.661,A 0.000,B 0.000,C 90.000,E1 154.921} C_DIS
LIN {X 0.165,Y -482.694,Z 303.647,A 0.000,B 0.000,C 90.000,E1 152.410} C_DIS
LIN {X -0.226,Y -488.364,Z 303.628,A 0.000,B 0.000,C 90.000,E1 149.076} C_DIS
LIN {X -0.164,Y -492.952,Z 303.615,A 0.000,B 0.000,C 90.000,E1 146.628} C_DIS
LIN {X 0.178,Y -496.597,Z 303.604,A 0.000,B 0.000,C 90.000,E1 144.769} C_DIS
LIN {X -0.089,Y -499.539,Z 303.596,A 0.000,B 0.000,C 90.000,E1 143.290} C_DIS
LIN {X -0.008,Y -502.288,Z 303.588,A 0.000,B 0.000,C 90.000,E1 141.778} C_DIS
LIN {X -0.161,Y -504.353,Z 303.581,A 0.000,B 0.000,C 90.000,E1 140.598} C_DIS
LIN {X 0.152,Y -505.743,Z 303.576,A 0.000,B 0.000,C 90.000,E1 139.666} C_DIS
LIN {X 0.051,Y -507.349,Z 303.569,A 0.000,B 0.000,C 90.000,E1 138.485} C_DIS
LIN {X 0.030,Y -508.319,Z 303.564,A 0.000,B 0.000,C 90.000,E1 137.595} C_DIS
LIN {X -0.075,Y -509.227,Z 303.558,A 0.000,B 0.000,C 90.000,E1 136.419} C_DIS
LIN {X 0.304,Y -509.626,Z 303.553,A 0.000,B 0.000,C 90.000,E1 135.486} C_DIS
LIN {X -0.042,Y -509.759,Z 303.548,A 0.000,B 0.000,C 90.000,E1 134.636} C_DIS
LIN {X -0.016,Y -509.644,Z 303.543,A 0.000,B 0.000,C 90.000,E1 133.743} C_DIS
LIN {X 0.104,Y -509.461,Z 303.540,A 0.000,B 0.000,C 90.000,E1 133.137} C_DIS
LIN {X 0.139,Y -508.892,Z 303.535,A 0.000,B 0.000,C 90.000,E1 132.243} C_DIS
LIN {X -0.203,Y -508.087,Z 303.530,A 0.000,B 0.000,C 90.000,E1 131.391} C_DIS
LIN {X -0.043,Y -506.344,Z 303.522,A 0.000,B 0.000,C 90.000,E1 129.886} C_DIS
LIN {X 0.076,Y -504.324,Z 303.513,A 0.000,B 0.000,C 90.000,E1 128.382} C_DIS
LIN {X -0.055,Y -502.640,Z 303.507,A 0.000,B 0.000,C 90.000,E1 127.202} C_DIS
LIN {X -0.233,Y -500.329,Z 303.498,A 0.000,B 0.000,C 90.000,E1 125.724} C_DIS
LIN {X 0.090,Y -498.187,Z 303.492,A 0.000,B 0.000,C 90.000,E1 124.485} C_DIS
LIN {X 0.243,Y -495.400,Z 303.483,A 0.000,B 0.000,C 90.000,E1 122.959} C_DIS
LIN {X -0.089,Y -491.830,Z 303.473,A 0.000,B 0.000,C 90.000,E1 121.180} C_DIS
LIN {X 0.085,Y -487.619,Z 303.461,A 0.000,B 0.000,C 90.000,E1 119.027} C_DIS
LIN {X -0.063,Y -484.537,Z 303.453,A 0.000,B 0.000,C 90.000,E1 117.513} C_DIS
LIN {X -0.069,Y -481.465,Z 303.444,A 0.000,B 0.000,C 90.000,E1 115.976} C_DIS
LIN {X -0.155,Y -477.793,Z 303.434,A 0.000,B 0.000,C 90.000,E1 114.131} C_DIS
LIN {X -0.119,Y -473.555,Z 303.422,A 0.000,B 0.000,C 90.000,E1 111.950} C_DIS
LIN {X -0.057,Y -470.002,Z 303.411,A 0.000,B 0.000,C 90.000,E1 110.066} C_DIS
LIN {X -0.009,Y -467.063,Z 303.403,A 0.000,B 0.000,C 90.000,E1 108.489} C_DIS
LIN {X 0.132,Y -463.740,Z 303.392,A 0.000,B 0.000,C 90.000,E1 106.567} C_DIS
LIN {X 0.092,Y -463.742,Z 303.392,A 0.000,B 0.000,C 90.000,E1 106.567} C_DIS
LIN {X 0.021,Y -467.495,Z 303.383,A 0.000,B 0.000,C 90.000,E1 105.009} C_DIS
LIN {X -0.174,Y -468.087,Z 303.382,A 0.000,B 0.000,C 90.000,E1 104.717} C_DIS
LIN {X -0.036,Y -475.741,Z 303.357,A 0.000,B 0.000,C 90.000,E1 100.310} C_DIS
LIN {X -0.199,Y -476.278,Z 303.356,A 0.000,B 0.000,C 90.000,E1 100.018} C_DIS
LIN {X 0.218,Y -481.743,Z 303.331,A 0.000,B 0.000,C 90.000,E1 95.625} C_DIS
LIN {X 0.065,Y -482.159,Z 303.330,A 0.000,B 0.000,C 90.000,E1 95.334} C_DIS
LIN {X -0.180,Y -485.538,Z 303.304,A 0.000,B 0.000,C 90.000,E1 90.745} C_DIS
LIN {X 0.027,Y -486.305,Z 303.282,A 0.000,B 0.000,C 90.000,E1 86.731} C_DIS
LIN {X 0.162,Y -486.325,Z 303.279,A 0.000,B 0.000,C 90.000,E1 86.102} C_DIS
LIN {X 0.235,Y -484.630,Z 303.253,A 0.000,B 0.000,C 90.000,E1 81.489} C_DIS
LIN {X 0.114,Y -480.558,Z 303.227,A 0.000,B 0.000,C 90.000,E1 76.881} C_DIS
LIN {X 0.150,Y -475.098,Z 303.205,A 0.000,B 0.000,C 90.000,E1 72.960} C_DIS
LIN {X 0.064,Y -481.417,Z 303.191,A 0.000,B 0.000,C 90.000,E1 70.369} C_DIS
LIN {X 0.062,Y -484.639,Z 303.184,A 0.000,B 0.000,C 90.000,E1 69.135} C_DIS
LIN {X -0.048,Y -488.832,Z 303.176,A 0.000,B 0.000,C 90.000,E1 67.614} C_DIS
LIN {X -0.086,Y -494.719,Z 303.164,A 0.000,B 0.000,C 90.000,E1 65.485} C_DIS
LIN {X -0.206,Y -500.694,Z 303.152,A 0.000,B 0.000,C 90.000,E1 63.384} C_DIS
LIN {X -0.014,Y -505.919,Z 303.142,A 0.000,B 0.000,C 90.000,E1 61.563} C_DIS
LIN {X 0.190,Y -512.019,Z 303.130,A 0.000,B 0.000,C 90.000,E1 59.459} C_DIS
LIN {X 0.010,Y -517.184,Z 303.121,A 0.000,B 0.000,C 90.000,E1 57.709} C_DIS
LIN {X 0.275,Y -521.438,Z 303.113,A 0.000,B 0.000,C 90.000,E1 56.215} C_DIS
LIN {X 0.177,Y -525.587,Z 303.104,A 0.000,B 0.000,C 90.000,E1 54.769} C_DIS
LIN {X 0.026,Y -529.398,Z 303.096,A 0.000,B 0.000,C 90.000,E1 53.336} C_DIS
LIN {X -0.029,Y -531.501,Z 303.092,A 0.000,B 0.000,C 90.000,E1 52.477} C_DIS
LIN {X -0.074,Y -534.189,Z 303.085,A 0.000,B 0.000,C 90.000,E1 51.331} C_DIS
LIN {X -0.160,Y -537.175,Z 303.077,A 0.000,B 0.000,C 90.000,E1 49.908} C_DIS
LIN {X 0.201,Y -538.764,Z 303.072,A 0.000,B 0.000,C 90.000,E1 49.013} C_DIS
LIN {X -0.221,Y -540.713,Z 303.066,A 0.000,B 0.000,C 90.000,E1 47.919} C_DIS
LIN {X 0.155,Y -542.426,Z 303.060,A 0.000,B 0.000,C 90.000,E1 46.743} C_DIS
LIN {X -0.215,Y -543.788,Z 303.054,A 0.000,B 0.000,C 90.000,E1 45.648} C_DIS
LIN {X 0.190,Y -544.560,Z 303.049,A 0.000,B 0.000,C 90.000,E1 44.757} C_DIS
LIN {X 0.226,Y -545.380,Z 303.043,A 0.000,B 0.000,C 90.000,E1 43.623} C_DIS
LIN {X -0.106,Y -545.964,Z 303.036,A 0.000,B 0.000,C 90.000,E1 42.528} C_DIS
LIN {X -0.022,Y -546.410,Z 303.030,A 0.000,B 0.000,C 90.000,E1 41.391} C_DIS
LIN {X 0.070,Y -546.557,Z 303.024,A 0.000,B 0.000,C 90.000,E1 40.253} C_DIS
LIN {X 0.119,Y -546.555,Z 303.019,A 0.000,B 0.000,C 90.000,E1 39.402} C_DIS
LIN {X 0.244,Y -546.350,Z 303.014,A 0.000,B 0.000,C 90.000,E1 38.543} C_DIS
LIN {X -0.018,Y -545.772,Z 303.008,A 0.000,B 0.000,C 90.000,E1 37.443} C_DIS
LIN {X 0.180,Y -544.808,Z 303.000,A 0.000,B 0.000,C 90.000,E1 36.011} C_DIS
LIN {X 0.072,Y -543.415,Z 302.991,A 0.000,B 0.000,C 90.000,E1 34.326} C_DIS
LIN {X 0.059,Y -542.135,Z 302.983,A 0.000,B 0.000,C 90.000,E1 32.911} C_DIS
LIN {X -0.213,Y -539.947,Z 302.970,A 0.000,B 0.000,C 90.000,E1 30.669} C_DIS
LIN {X 0.176,Y -538.600,Z 302.962,A 0.000,B 0.000,C 90.000,E1 29.205} C_DIS
LIN {X -0.276,Y -536.665,Z 302.951,A 0.000,B 0.000,C 90.000,E1 27.257} C_DIS
LIN {X -0.256,Y -534.967,Z 302.942,A 0.000,B 0.000,C 90.000,E1 25.540} C_DIS
LIN {X 0.011,Y -533.613,Z 302.934,A 0.000,B 0.000,C 90.000,E1 24.079} C_DIS
LIN {X -0.070,Y -531.894,Z 302.923,A 0.000,B 0.000,C 90.000,E1 22.078} C_DIS
LIN {X 0.096,Y -530.162,Z 302.910,A 0.000,B 0.000,C 90.000,E1 19.758} C_DIS
LIN {X -0.150,Y -529.042,Z 302.900,A 0.000,B 0.000,C 90.000,E1 18.055} C_DIS
LIN {X -0.089,Y -528.030,Z 302.891,A 0.000,B 0.000,C 90.000,E1 16.315} C_DIS
LIN {X -0.172,Y -527.211,Z 302.879,A 0.000,B 0.000,C 90.000,E1 14.300} C_DIS
LIN {X 0.138,Y -526.535,Z 302.867,A 0.000,B 0.000,C 90.000,E1 11.951} C_DIS
LIN {X -0.178,Y -526.121,Z 302.852,A 0.000,B 0.000,C 90.000,E1 9.378} C_DIS
LIN {X -0.212,Y -526.159,Z 302.841,A 0.000,B 0.000,C 90.000,E1 7.352} C_DIS
LIN {X 0.216,Y -526.506,Z 302.829,A 0.000,B 0.000,C 90.000,E1 5.277} C_DIS
LIN {X 0.042,Y -527.301,Z 302.817,A 0.000,B 0.000,C 90.000,E1 2.980} C_DIS
LIN {X -0.082,Y -527.974,Z 302.809,A 0.000,B 0.000,C 90.000,E1 1.547} C_DIS
LIN {X 0.057,Y -530.642,Z 302.786,A 0.000,B 0.000,C 90.000,E1 357.478} C_DIS
LIN {X -0.001,Y -532.456,Z 302.775,A 0.000,B 0.000,C 90.000,E1 355.469} C_DIS
LIN {X 0.223,Y -537.434,Z 302.753,A 0.000,B 0.000,C 90.000,E1 351.432} C_DIS
LIN {X -0.154,Y -543.366,Z 302.735,A 0.000,B 0.000,C 90.000,E1 348.342} C_DIS
LIN {X 0.042,Y -548.806,Z 302.723,A 0.000,B 0.000,C 90.000,E1 346.061} C_DIS
LIN {X 0.264,Y -554.675,Z 302.710,A 0.000,B 0.000,C 90.000,E1 343.795} C_DIS
LIN {X 0.130,Y -560.880,Z 302.698,A 0.000,B 0.000,C 90.000,E1 341.583} C_DIS
LIN {X 0.188,Y -566.600,Z 302.687,A 0.000,B 0.000,C 90.000,E1 339.645} C_DIS
LIN {X -0.089,Y -571.822,Z 302.678,A 0.000,B 0.000,C 90.000,E1 338.028} C_DIS
LIN {X -0.086,Y -576.348,Z 302.670,A 0.000,B 0.000,C 90.000,E1 336.666} C_DIS
LIN {X -0.017,Y -580.894,Z 302.663,A 0.000,B 0.000,C 90.000,E1 335.305} C_DIS
LIN {X -0.146,Y -587.574,Z 302.652,A 0.000,B 0.000,C 90.000,E1 333.435} C_DIS
LIN {X -0.175,Y -592.324,Z 302.645,A 0.000,B 0.000,C 90.000,E1 332.103} C_DIS
LIN {X -0.379,Y -596.888,Z 302.638,A 0.000,B 0.000,C 90.000,E1 330.795} C_DIS
LIN {X -0.048,Y -603.275,Z 302.627,A 0.000,B 0.000,C 90.000,E1 328.918} C_DIS
LIN {X -0.064,Y -609.628,Z 302.617,A 0.000,B 0.000,C 90.000,E1 327.089} C_DIS
LIN {X 0.058,Y -616.035,Z 302.607,A 0.000,B 0.000,C 90.000,E1 325.261} C_DIS
LIN {X -0.077,Y -619.749,Z 302.601,A 0.000,B 0.000,C 90.000,E1 324.242} C_DIS
LIN {X -0.188,Y -623.965,Z 302.594,A 0.000,B 0.000,C 90.000,E1 322.970} C_DIS
LIN {X 0.292,Y -627.069,Z 302.589,A 0.000,B 0.000,C 90.000,E1 321.904} C_DIS
LIN {X -0.345,Y -631.590,Z 302.580,A 0.000,B 0.000,C 90.000,E1 320.436} C_DIS
LIN {X 0.031,Y -635.390,Z 302.573,A 0.000,B 0.000,C 90.000,E1 319.138} C_DIS
LIN {X -0.326,Y -638.342,Z 302.567,A 0.000,B 0.000,C 90.000,E1 318.162} C_DIS
LIN {X -0.155,Y -644.782,Z 302.555,A 0.000,B 0.000,C 90.000,E1 315.891} C_DIS
LIN {X -0.036,Y -648.495,Z 302.548,A 0.000,B 0.000,C 90.000,E1 314.636} C_DIS
LIN {X 0.199,Y -651.318,Z 302.542,A 0.000,B 0.000,C 90.000,E1 313.623} C_DIS
LIN {X -0.006,Y -654.644,Z 302.536,A 0.000,B 0.000,C 90.000,E1 312.405} C_DIS
LIN {X -0.168,Y -657.181,Z 302.530,A 0.000,B 0.000,C 90.000,E1 311.434} C_DIS
LIN {X 0.220,Y -660.046,Z 302.523,A 0.000,B 0.000,C 90.000,E1 310.172} C_DIS
LIN {X -0.266,Y -662.595,Z 302.517,A 0.000,B 0.000,C 90.000,E1 308.991} C_DIS
LIN {X -0.278,Y -664.453,Z 302.511,A 0.000,B 0.000,C 90.000,E1 308.016} C_DIS
LIN {X -0.151,Y -666.079,Z 302.506,A 0.000,B 0.000,C 90.000,E1 307.030} C_DIS
LIN {X 0.401,Y -667.368,Z 302.500,A 0.000,B 0.000,C 90.000,E1 306.011} C_DIS
LIN {X 0.063,Y -668.144,Z 302.496,A 0.000,B 0.000,C 90.000,E1 305.311} C_DIS
LIN {X -0.268,Y -668.554,Z 302.492,A 0.000,B 0.000,C 90.000,E1 304.612} C_DIS
LIN {X -0.087,Y -668.842,Z 302.487,A 0.000,B 0.000,C 90.000,E1 303.627} C_DIS
LIN {X 0.141,Y -668.820,Z 302.483,A 0.000,B 0.000,C 90.000,E1 302.880} C_DIS
LIN {X 0.371,Y -668.577,Z 302.479,A 0.000,B 0.000,C 90.000,E1 302.133} C_DIS
LIN {X 0.099,Y -668.237,Z 302.476,A 0.000,B 0.000,C 90.000,E1 301.671} C_DIS
LIN {X 0.322,Y -667.351,Z 302.472,A 0.000,B 0.000,C 90.000,E1 300.924} C_DIS
LIN {X 0.046,Y -666.636,Z 302.469,A 0.000,B 0.000,C 90.000,E1 300.463} C_DIS
LIN {X 0.062,Y -664.775,Z 302.464,A 0.000,B 0.000,C 90.000,E1 299.489} C_DIS
LIN {X -0.063,Y -662.069,Z 302.457,A 0.000,B 0.000,C 90.000,E1 298.281} C_DIS
LIN {X -0.108,Y -659.737,Z 302.452,A 0.000,B 0.000,C 90.000,E1 297.308} C_DIS
LIN {X -0.234,Y -655.978,Z 302.444,A 0.000,B 0.000,C 90.000,E1 295.848} C_DIS
LIN {X 0.114,Y -654.066,Z 302.439,A 0.000,B 0.000,C 90.000,E1 295.079} C_DIS
LIN {X 0.368,Y -650.704,Z 302.433,A 0.000,B 0.000,C 90.000,E1 293.823} C_DIS
LIN {X -0.369,Y -645.974,Z 302.423,A 0.000,B 0.000,C 90.000,E1 292.153} C_DIS
LIN {X 0.107,Y -642.685,Z 302.416,A 0.000,B 0.000,C 90.000,E1 290.865} C_DIS
LIN {X -0.249,Y -638.807,Z 302.408,A 0.000,B 0.000,C 90.000,E1 289.396} C_DIS
LIN {X 0.155,Y -633.921,Z 302.397,A 0.000,B 0.000,C 90.000,E1 287.347} C_DIS
LIN {X 0.023,Y -628.465,Z 302.382,A 0.000,B 0.000,C 90.000,E1 284.828} C_DIS
LIN {X 0.231,Y -623.418,Z 302.367,A 0.000,B 0.000,C 90.000,E1 282.007} C_DIS
LIN {X 0.022,Y -619.529,Z 302.351,A 0.000,B 0.000,C 90.000,E1 279.208} C_DIS
LIN {X -0.233,Y -616.519,Z 302.334,A 0.000,B 0.000,C 90.000,E1 276.144} C_DIS
LIN {X -0.125,Y -614.816,Z 302.317,A 0.000,B 0.000,C 90.000,E1 273.037} C_DIS
LIN {X 0.124,Y -614.319,Z 302.304,A 0.000,B 0.000,C 90.000,E1 270.688} C_DIS
LIN {X 0.023,Y -614.969,Z 302.284,A 0.000,B 0.000,C 90.000,E1 267.078} C_DIS
LIN {X -0.193,Y -617.183,Z 302.265,A 0.000,B 0.000,C 90.000,E1 263.742} C_DIS
LIN {X -0.272,Y -619.429,Z 302.252,A 0.000,B 0.000,C 90.000,E1 261.432} C_DIS
LIN {X 0.079,Y -621.315,Z 302.244,A 0.000,B 0.000,C 90.000,E1 259.859} C_DIS
LIN {X 0.262,Y -623.819,Z 302.234,A 0.000,B 0.000,C 90.000,E1 258.049} C_DIS
LIN {X -0.316,Y -625.722,Z 302.227,A 0.000,B 0.000,C 90.000,E1 256.825} C_DIS
LIN {X 0.031,Y -627.614,Z 302.220,A 0.000,B 0.000,C 90.000,E1 255.519} C_DIS
LIN {X -0.159,Y -629.061,Z 302.214,A 0.000,B 0.000,C 90.000,E1 254.519} C_DIS
LIN {X 0.028,Y -629.887,Z 302.210,A 0.000,B 0.000,C 90.000,E1 253.740} C_DIS
LIN {X 0.034,Y -630.754,Z 302.204,A 0.000,B 0.000,C 90.000,E1 252.725} C_DIS
LIN {X 0.241,Y -631.397,Z 302.200,A 0.000,B 0.000,C 90.000,E1 251.945} C_DIS
LIN {X -0.148,Y -631.917,Z 302.196,A 0.000,B 0.000,C 90.000,E1 251.221} C_DIS
LIN {X 0.077,Y -632.266,Z 302.190,A 0.000,B 0.000,C 90.000,E1 250.188} C_DIS
LIN {X -0.289,Y -632.254,Z 302.184,A 0.000,B 0.000,C 90.000,E1 249.209} C_DIS
LIN {X 0.166,Y -631.848,Z 302.179,A 0.000,B 0.000,C 90.000,E1 248.156} C_DIS
LIN {X -0.209,Y -630.994,Z 302.173,A 0.000,B 0.000,C 90.000,E1 247.177} C_DIS
LIN {X -0.129,Y -630.083,Z 302.169,A 0.000,B 0.000,C 90.000,E1 246.410} C_DIS
LIN {X 0.290,Y -628.436,Z 302.163,A 0.000,B 0.000,C 90.000,E1 245.357} C_DIS
LIN {X 0.355,Y -627.006,Z 302.159,A 0.000,B 0.000,C 90.000,E1 244.588} C_DIS
LIN {X 0.134,Y -625.339,Z 302.155,A 0.000,B 0.000,C 90.000,E1 243.845} C_DIS
LIN {X 0.173,Y -622.749,Z 302.149,A 0.000,B 0.000,C 90.000,E1 242.820} C_DIS
LIN {X -0.372,Y -620.692,Z 302.145,A 0.000,B 0.000,C 90.000,E1 242.103} C_DIS
LIN {X -0.115,Y -617.002,Z 302.138,A 0.000,B 0.000,C 90.000,E1 240.795} C_DIS
LIN {X 0.073,Y -613.209,Z 302.131,A 0.000,B 0.000,C 90.000,E1 239.488} C_DIS
LIN {X -0.023,Y -609.284,Z 302.123,A 0.000,B 0.000,C 90.000,E1 238.201} C_DIS
LIN {X -0.177,Y -605.327,Z 302.116,A 0.000,B 0.000,C 90.000,E1 236.914} C_DIS
LIN {X 0.185,Y -600.603,Z 302.107,A 0.000,B 0.000,C 90.000,E1 235.308} C_DIS
LIN {X -0.023,Y -597.324,Z 302.102,A 0.000,B 0.000,C 90.000,E1 234.276} C_DIS
LIN {X 0.039,Y -592.009,Z 302.093,A 0.000,B 0.000,C 90.000,E1 232.683} C_DIS
LIN {X -0.070,Y -585.098,Z 302.081,A 0.000,B 0.000,C 90.000,E1 230.561} C_DIS
LIN {X 0.105,Y -579.864,Z 302.072,A 0.000,B 0.000,C 90.000,E1 228.933} C_DIS
LIN {X -0.047,Y -573.218,Z 302.060,A 0.000,B 0.000,C 90.000,E1 226.782} C_DIS
LIN {X -0.204,Y -568.111,Z 302.051,A 0.000,B 0.000,C 90.000,E1 225.162} C_DIS
LIN {X 0.013,Y -562.239,Z 302.040,A 0.000,B 0.000,C 90.000,E1 223.218} C_DIS
LIN {X 0.066,Y -557.263,Z 302.031,A 0.000,B 0.000,C 90.000,E1 221.553} C_DIS
LIN {X -0.335,Y -551.372,Z 302.020,A 0.000,B 0.000,C 90.000,E1 219.644} C_DIS
LIN {X -0.047,Y -545.383,Z 302.009,A 0.000,B 0.000,C 90.000,E1 217.649} C_DIS
LIN {X 0.100,Y -542.043,Z 302.003,A 0.000,B 0.000,C 90.000,E1 216.503} C_DIS
LIN {X -0.071,Y -535.442,Z 301.990,A 0.000,B 0.000,C 90.000,E1 214.246} C_DIS
LIN {X 0.151,Y -529.043,Z 301.978,A 0.000,B 0.000,C 90.000,E1 211.926} C_DIS
LIN {X 0.096,Y -523.024,Z 301.965,A 0.000,B 0.000,C 90.000,E1 209.617} C_DIS
LIN {X -0.041,Y -517.904,Z 301.953,A 0.000,B 0.000,C 90.000,E1 207.590} C_DIS
LIN {X -0.088,Y -513.005,Z 301.942,A 0.000,B 0.000,C 90.000,E1 205.540} C_DIS
LIN {X -0.123,Y -509.069,Z 301.932,A 0.000,B 0.000,C 90.000,E1 203.770} C_DIS
LIN {X 0.110,Y -504.667,Z 301.920,A 0.000,B 0.000,C 90.000,E1 201.663} C_DIS
LIN {X -0.032,Y -501.084,Z 301.910,A 0.000,B 0.000,C 90.000,E1 199.885} C_DIS
LIN {X 0.069,Y -496.047,Z 301.895,A 0.000,B 0.000,C 90.000,E1 197.166} C_DIS
LIN {X 0.184,Y -491.453,Z 301.880,A 0.000,B 0.000,C 90.000,E1 194.426} C_DIS
LIN {X -0.122,Y -489.128,Z 301.872,A 0.000,B 0.000,C 90.000,E1 192.939} C_DIS
LIN {X 0.025,Y -485.972,Z 301.860,A 0.000,B 0.000,C 90.000,E1 190.782} C_DIS
LIN {X 0.091,Y -483.077,Z 301.848,A 0.000,B 0.000,C 90.000,E1 188.624} C_DIS
LIN {X 0.074,Y -480.790,Z 301.838,A 0.000,B 0.000,C 90.000,E1 186.777} C_DIS
LIN {X -0.207,Y -478.239,Z 301.826,A 0.000,B 0.000,C 90.000,E1 184.645} C_DIS
LIN {X -0.214,Y -476.663,Z 301.817,A 0.000,B 0.000,C 90.000,E1 183.094} C_DIS
LIN {X 0.196,Y -475.156,Z 301.808,A 0.000,B 0.000,C 90.000,E1 181.489} C_DIS
LIN {X -0.229,Y -472.635,Z 301.789,A 0.000,B 0.000,C 90.000,E1 178.108} C_DIS
LIN {X 0.184,Y -471.343,Z 301.774,A 0.000,B 0.000,C 90.000,E1 175.241} C_DIS
LIN {X -0.047,Y -470.673,Z 301.760,A 0.000,B 0.000,C 90.000,E1 172.761} C_DIS
LIN {X 0.203,Y -470.394,Z 301.749,A 0.000,B 0.000,C 90.000,E1 170.849} C_DIS
LIN {X -0.023,Y -470.385,Z 301.739,A 0.000,B 0.000,C 90.000,E1 168.993} C_DIS
LIN {X -0.011,Y -471.195,Z 301.718,A 0.000,B 0.000,C 90.000,E1 165.227} C_DIS
LIN {X 0.144,Y -472.202,Z 301.706,A 0.000,B 0.000,C 90.000,E1 163.015} C_DIS
LIN {X -0.160,Y -473.882,Z 301.692,A 0.000,B 0.000,C 90.000,E1 160.550} C_DIS
LIN {X 0.061,Y -475.804,Z 301.678,A 0.000,B 0.000,C 90.000,E1 158.028} C_DIS
LIN {X 0.072,Y -478.621,Z 301.662,A 0.000,B 0.000,C 90.000,E1 155.229} C_DIS
LIN {X -0.054,Y -481.409,Z 301.650,A 0.000,B 0.000,C 90.000,E1 153.076} C_DIS
LIN {X -0.081,Y -486.216,Z 301.633,A 0.000,B 0.000,C 90.000,E1 149.999} C_DIS
LIN {X 0.190,Y -488.413,Z 301.627,A 0.000,B 0.000,C 90.000,E1 148.742} C_DIS
LIN {X 0.000,Y -492.391,Z 301.615,A 0.000,B 0.000,C 90.000,E1 146.628} C_DIS
LIN {X 0.068,Y -495.397,Z 301.606,A 0.000,B 0.000,C 90.000,E1 145.102} C_DIS
LIN {X -0.215,Y -498.290,Z 301.598,A 0.000,B 0.000,C 90.000,E1 143.623} C_DIS
LIN {X -0.027,Y -500.508,Z 301.591,A 0.000,B 0.000,C 90.000,E1 142.396} C_DIS
LIN {X 0.076,Y -503.069,Z 301.583,A 0.000,B 0.000,C 90.000,E1 140.884} C_DIS
LIN {X 0.050,Y -504.529,Z 301.578,A 0.000,B 0.000,C 90.000,E1 139.989} C_DIS
LIN {X 0.261,Y -506.163,Z 301.571,A 0.000,B 0.000,C 90.000,E1 138.771} C_DIS
LIN {X -0.111,Y -507.184,Z 301.566,A 0.000,B 0.000,C 90.000,E1 137.919} C_DIS
LIN {X -0.100,Y -507.976,Z 301.561,A 0.000,B 0.000,C 90.000,E1 137.025} C_DIS
LIN {X -0.108,Y -508.555,Z 301.556,A 0.000,B 0.000,C 90.000,E1 136.134} C_DIS
LIN {X 0.016,Y -508.826,Z 301.553,A 0.000,B 0.000,C 90.000,E1 135.526} C_DIS
LIN {X -0.097,Y -508.959,Z 301.546,A 0.000,B 0.000,C 90.000,E1 134.352} C_DIS
LIN {X 0.149,Y -508.665,Z 301.540,A 0.000,B 0.000,C 90.000,E1 133.137} C_DIS
LIN {X -0.200,Y -508.120,Z 301.535,A 0.000,B 0.000,C 90.000,E1 132.285} C_DIS
LIN {X -0.174,Y -507.309,Z 301.530,A 0.000,B 0.000,C 90.000,E1 131.391} C_DIS
LIN {X -0.029,Y -505.577,Z 301.522,A 0.000,B 0.000,C 90.000,E1 129.886} C_DIS
LIN {X 0.075,Y -503.558,Z 301.513,A 0.000,B 0.000,C 90.000,E1 128.382} C_DIS
LIN {X -0.068,Y -501.848,Z 301.507,A 0.000,B 0.000,C 90.000,E1 127.202} C_DIS
LIN {X 0.146,Y -499.539,Z 301.498,A 0.000,B 0.000,C 90.000,E1 125.678} C_DIS
LIN {X 0.051,Y -497.385,Z 301.492,A 0.000,B 0.000,C 90.000,E1 124.485} C_DIS
LIN {X 0.191,Y -494.597,Z 301.483,A 0.000,B 0.000,C 90.000,E1 122.959} C_DIS
LIN {X 0.002,Y -491.622,Z 301.475,A 0.000,B 0.000,C 90.000,E1 121.465} C_DIS
LIN {X -0.007,Y -487.441,Z 301.463,A 0.000,B 0.000,C 90.000,E1 119.333} C_DIS
LIN {X 0.264,Y -484.386,Z 301.454,A 0.000,B 0.000,C 90.000,E1 117.769} C_DIS
LIN {X -0.188,Y -480.714,Z 301.444,A 0.000,B 0.000,C 90.000,E1 115.976} C_DIS
LIN {X 0.147,Y -477.056,Z 301.434,A 0.000,B 0.000,C 90.000,E1 114.079} C_DIS
LIN {X 0.168,Y -472.828,Z 301.422,A 0.000,B 0.000,C 90.000,E1 111.897} C_DIS
LIN {X -0.270,Y -468.759,Z 301.410,A 0.000,B 0.000,C 90.000,E1 109.758} C_DIS
LIN {X 0.030,Y -463.533,Z 301.393,A 0.000,B 0.000,C 90.000,E1 106.804} C_DIS
LIN {X 0.007,Y -463.408,Z 301.393,A 0.000,B 0.000,C 90.000,E1 106.732} C_DIS
LIN {X -0.033,Y -463.406,Z 301.393,A 0.000,B 0.000,C 90.000,E1 106.732} C_DIS
LIN {X -0.178,Y -467.556,Z 301.383,A 0.000,B 0.000,C 90.000,E1 105.009} C_DIS
LIN {X 0.006,Y -468.571,Z 301.380,A 0.000,B 0.000,C 90.000,E1 104.356} C_DIS
LIN {X 0.232,Y -475.791,Z 301.357,A 0.000,B 0.000,C 90.000,E1 100.254} C_DIS
LIN {X 0.070,Y -476.301,Z 301.355,A 0.000,B 0.000,C 90.000,E1 99.962} C_DIS
LIN {X 0.018,Y -481.782,Z 301.331,A 0.000,B 0.000,C 90.000,E1 95.625} C_DIS
LIN {X -0.135,Y -482.170,Z 301.330,A 0.000,B 0.000,C 90.000,E1 95.334} C_DIS
LIN {X -0.206,Y -485.303,Z 301.306,A 0.000,B 0.000,C 90.000,E1 91.031} C_DIS
LIN {X 0.104,Y -485.537,Z 301.304,A 0.000,B 0.000,C 90.000,E1 90.688} C_DIS
LIN {X -0.174,Y -486.317,Z 301.282,A 0.000,B 0.000,C 90.000,E1 86.731} C_DIS
LIN {X -0.040,Y -486.308,Z 301.278,A 0.000,B 0.000,C 90.000,E1 86.102} C_DIS
LIN {X 0.165,Y -484.696,Z 301.254,A 0.000,B 0.000,C 90.000,E1 81.781} C_DIS
LIN {X 0.034,Y -484.606,Z 301.253,A 0.000,B 0.000,C 90.000,E1 81.489} C_DIS
LIN {X -0.086,Y -480.539,Z 301.227,A 0.000,B 0.000,C 90.000,E1 76.881} C_DIS
LIN {X -0.160,Y -474.888,Z 301.204,A 0.000,B 0.000,C 90.000,E1 72.779} C_DIS
LIN {X -0.169,Y -482.412,Z 301.187,A 0.000,B 0.000,C 90.000,E1 69.752} C_DIS
LIN {X -0.106,Y -488.160,Z 301.175,A 0.000,B 0.000,C 90.000,E1 67.592} C_DIS
LIN {X 0.099,Y -494.024,Z 301.164,A 0.000,B 0.000,C 90.000,E1 65.433} C_DIS
LIN {X -0.046,Y -500.009,Z 301.152,A 0.000,B 0.000,C 90.000,E1 63.332} C_DIS
LIN {X 0.124,Y -505.245,Z 301.142,A 0.000,B 0.000,C 90.000,E1 61.513} C_DIS
LIN {X -0.137,Y -511.345,Z 301.130,A 0.000,B 0.000,C 90.000,E1 59.459} C_DIS
LIN {X 0.025,Y -517.358,Z 301.119,A 0.000,B 0.000,C 90.000,E1 57.375} C_DIS
LIN {X -0.143,Y -521.579,Z 301.111,A 0.000,B 0.000,C 90.000,E1 55.928} C_DIS
LIN {X -0.200,Y -524.919,Z 301.104,A 0.000,B 0.000,C 90.000,E1 54.769} C_DIS
LIN {X 0.059,Y -528.703,Z 301.096,A 0.000,B 0.000,C 90.000,E1 53.290} C_DIS
LIN {X -0.027,Y -531.487,Z 301.090,A 0.000,B 0.000,C 90.000,E1 52.145} C_DIS
LIN {X 0.264,Y -533.502,Z 301.085,A 0.000,B 0.000,C 90.000,E1 51.251} C_DIS
LIN {X 0.169,Y -536.505,Z 301.077,A 0.000,B 0.000,C 90.000,E1 49.828} C_DIS
LIN {X 0.125,Y -539.115,Z 301.069,A 0.000,B 0.000,C 90.000,E1 48.405} C_DIS
LIN {X -0.292,Y -540.888,Z 301.063,A 0.000,B 0.000,C 90.000,E1 47.310} C_DIS
LIN {X 0.077,Y -542.063,Z 301.058,A 0.000,B 0.000,C 90.000,E1 46.419} C_DIS
LIN {X -0.298,Y -543.362,Z 301.052,A 0.000,B 0.000,C 90.000,E1 45.324} C_DIS
LIN {X -0.278,Y -544.261,Z 301.045,A 0.000,B 0.000,C 90.000,E1 44.190} C_DIS
LIN {X 0.127,Y -544.803,Z 301.041,A 0.000,B 0.000,C 90.000,E1 43.299} C_DIS
LIN {X 0.203,Y -545.588,Z 301.031,A 0.000,B 0.000,C 90.000,E1 41.595} C_DIS
LIN {X 0.280,Y -545.755,Z 301.025,A 0.000,B 0.000,C 90.000,E1 40.458} C_DIS
LIN {X 0.009,Y -545.762,Z 301.019,A 0.000,B 0.000,C 90.000,E1 39.358} C_DIS
LIN {X -0.337,Y -545.661,Z 301.016,A 0.000,B 0.000,C 90.000,E1 38.830} C_DIS
LIN {X 0.118,Y -545.288,Z 301.011,A 0.000,B 0.000,C 90.000,E1 37.935} C_DIS
LIN {X 0.268,Y -544.614,Z 301.005,A 0.000,B 0.000,C 90.000,E1 36.790} C_DIS
LIN {X 0.091,Y -543.802,Z 300.998,A 0.000,B 0.000,C 90.000,E1 35.678} C_DIS
LIN {X -0.060,Y -542.661,Z 300.990,A 0.000,B 0.000,C 90.000,E1 34.278} C_DIS
LIN {X -0.240,Y -541.389,Z 300.983,A 0.000,B 0.000,C 90.000,E1 32.880} C_DIS
LIN {X -0.087,Y -539.182,Z 300.970,A 0.000,B 0.000,C 90.000,E1 30.590} C_DIS
LIN {X 0.021,Y -537.826,Z 300.962,A 0.000,B 0.000,C 90.000,E1 29.155} C_DIS
LIN {X 0.281,Y -535.856,Z 300.951,A 0.000,B 0.000,C 90.000,E1 27.129} C_DIS
LIN {X -0.002,Y -533.894,Z 300.940,A 0.000,B 0.000,C 90.000,E1 25.155} C_DIS
LIN {X -0.163,Y -531.544,Z 300.925,A 0.000,B 0.000,C 90.000,E1 22.589} C_DIS
LIN {X 0.002,Y -529.849,Z 300.914,A 0.000,B 0.000,C 90.000,E1 20.556} C_DIS
LIN {X 0.061,Y -529.310,Z 300.909,A 0.000,B 0.000,C 90.000,E1 19.685} C_DIS
LIN {X -0.204,Y -527.960,Z 300.898,A 0.000,B 0.000,C 90.000,E1 17.692} C_DIS
LIN {X 0.160,Y -527.258,Z 300.892,A 0.000,B 0.000,C 90.000,E1 16.496} C_DIS
LIN {X 0.077,Y -526.292,Z 300.879,A 0.000,B 0.000,C 90.000,E1 14.189} C_DIS
LIN {X -0.036,Y -525.564,Z 300.866,A 0.000,B 0.000,C 90.000,E1 11.883} C_DIS
LIN {X 0.012,Y -525.153,Z 300.853,A 0.000,B 0.000,C 90.000,E1 9.557} C_DIS
LIN {X -0.015,Y -525.160,Z 300.839,A 0.000,B 0.000,C 90.000,E1 6.947} C_DIS
LIN {X -0.187,Y -525.498,Z 300.827,A 0.000,B 0.000,C 90.000,E1 4.935} C_DIS
LIN {X -0.228,Y -525.693,Z 300.823,A 0.000,B 0.000,C 90.000,E1 4.069} C_DIS
LIN {X 0.177,Y -526.251,Z 300.816,A 0.000,B 0.000,C 90.000,E1 2.865} C_DIS
LIN {X 0.035,Y -526.884,Z 300.808,A 0.000,B 0.000,C 90.000,E1 1.432} C_DIS
LIN {X 0.046,Y -529.223,Z 300.788,A 0.000,B 0.000,C 90.000,E1 357.764} C_DIS
LIN {X -0.065,Y -531.269,Z 300.775,A 0.000,B 0.000,C 90.000,E1 355.469} C_DIS
LIN {X -0.225,Y -538.620,Z 300.745,A 0.000,B 0.000,C 90.000,E1 350.038} C_DIS
LIN {X -0.037,Y -547.603,Z 300.723,A 0.000,B 0.000,C 90.000,E1 346.047} C_DIS
LIN {X 0.015,Y -553.383,Z 300.710,A 0.000,B 0.000,C 90.000,E1 343.795} C_DIS
LIN {X -0.158,Y -559.599,Z 300.698,A 0.000,B 0.000,C 90.000,E1 341.583} C_DIS
LIN {X 0.268,Y -564.506,Z 300.688,A 0.000,B 0.000,C 90.000,E1 339.880} C_DIS
LIN {X -0.258,Y -569.728,Z 300.679,A 0.000,B 0.000,C 90.000,E1 338.284} C_DIS
LIN {X -0.298,Y -574.250,Z 300.672,A 0.000,B 0.000,C 90.000,E1 336.922} C_DIS
LIN {X 0.208,Y -580.613,Z 300.661,A 0.000,B 0.000,C 90.000,E1 334.973} C_DIS
LIN {X -0.057,Y -586.382,Z 300.652,A 0.000,B 0.000,C 90.000,E1 333.384} C_DIS
LIN {X 0.165,Y -591.148,Z 300.645,A 0.000,B 0.000,C 90.000,E1 332.025} C_DIS
LIN {X -0.050,Y -595.726,Z 300.637,A 0.000,B 0.000,C 90.000,E1 330.717} C_DIS
LIN {X -0.049,Y -602.069,Z 300.627,A 0.000,B 0.000,C 90.000,E1 328.869} C_DIS
LIN {X 0.163,Y -609.317,Z 300.615,A 0.000,B 0.000,C 90.000,E1 326.755} C_DIS
LIN {X 0.035,Y -613.939,Z 300.608,A 0.000,B 0.000,C 90.000,E1 325.468} C_DIS
LIN {X -0.179,Y -618.640,Z 300.601,A 0.000,B 0.000,C 90.000,E1 324.196} C_DIS
LIN {X -0.319,Y -622.904,Z 300.594,A 0.000,B 0.000,C 90.000,E1 322.924} C_DIS
LIN {X -0.353,Y -626.023,Z 300.588,A 0.000,B 0.000,C 90.000,E1 321.904} C_DIS
LIN {X -0.344,Y -629.074,Z 300.583,A 0.000,B 0.000,C 90.000,E1 320.884} C_DIS
LIN {X 0.348,Y -633.656,Z 300.574,A 0.000,B 0.000,C 90.000,E1 319.299} C_DIS
LIN {X -0.031,Y -636.679,Z 300.569,A 0.000,B 0.000,C 90.000,E1 318.324} C_DIS
LIN {X 0.090,Y -643.079,Z 300.556,A 0.000,B 0.000,C 90.000,E1 316.053} C_DIS
LIN {X -0.339,Y -647.536,Z 300.548,A 0.000,B 0.000,C 90.000,E1 314.595} C_DIS
LIN {X -0.164,Y -651.010,Z 300.541,A 0.000,B 0.000,C 90.000,E1 313.338} C_DIS
LIN {X 0.027,Y -654.933,Z 300.533,A 0.000,B 0.000,C 90.000,E1 311.838} C_DIS
LIN {X -0.078,Y -657.329,Z 300.527,A 0.000,B 0.000,C 90.000,E1 310.862} C_DIS
LIN {X -0.184,Y -660.061,Z 300.520,A 0.000,B 0.000,C 90.000,E1 309.644} C_DIS
LIN {X -0.227,Y -662.021,Z 300.515,A 0.000,B 0.000,C 90.000,E1 308.669} C_DIS
LIN {X 0.269,Y -663.779,Z 300.509,A 0.000,B 0.000,C 90.000,E1 307.649} C_DIS
LIN {X -0.108,Y -664.952,Z 300.505,A 0.000,B 0.000,C 90.000,E1 306.950} C_DIS
LIN {X 0.034,Y -666.232,Z 300.500,A 0.000,B 0.000,C 90.000,E1 305.964} C_DIS
LIN {X 0.074,Y -666.965,Z 300.496,A 0.000,B 0.000,C 90.000,E1 305.231} C_DIS
LIN {X -0.142,Y -667.395,Z 300.490,A 0.000,B 0.000,C 90.000,E1 304.278} C_DIS
LIN {X 0.447,Y -667.551,Z 300.486,A 0.000,B 0.000,C 90.000,E1 303.499} C_DIS
LIN {X -0.258,Y -667.507,Z 300.482,A 0.000,B 0.000,C 90.000,E1 302.832} C_DIS
LIN {X -0.036,Y -667.241,Z 300.478,A 0.000,B 0.000,C 90.000,E1 302.084} C_DIS
LIN {X 0.037,Y -666.829,Z 300.476,A 0.000,B 0.000,C 90.000,E1 301.592} C_DIS
LIN {X -0.099,Y -665.918,Z 300.472,A 0.000,B 0.000,C 90.000,E1 300.875} C_DIS
LIN {X 0.099,Y -664.714,Z 300.467,A 0.000,B 0.000,C 90.000,E1 300.129} C_DIS
LIN {X 0.091,Y -662.680,Z 300.462,A 0.000,B 0.000,C 90.000,E1 299.155} C_DIS
LIN {X 0.063,Y -660.474,Z 300.457,A 0.000,B 0.000,C 90.000,E1 298.180} C_DIS
LIN {X 0.008,Y -658.142,Z 300.451,A 0.000,B 0.000,C 90.000,E1 297.206} C_DIS
LIN {X 0.035,Y -654.996,Z 300.444,A 0.000,B 0.000,C 90.000,E1 295.976} C_DIS
LIN {X -0.388,Y -652.411,Z 300.439,A 0.000,B 0.000,C 90.000,E1 295.027} C_DIS
LIN {X -0.153,Y -649.057,Z 300.432,A 0.000,B 0.000,C 90.000,E1 293.770} C_DIS
LIN {X -0.076,Y -644.338,Z 300.422,A 0.000,B 0.000,C 90.000,E1 292.025} C_DIS
LIN {X -0.230,Y -641.023,Z 300.415,A 0.000,B 0.000,C 90.000,E1 290.791} C_DIS
LIN {X -0.203,Y -636.549,Z 300.406,A 0.000,B 0.000,C 90.000,E1 289.033} C_DIS
LIN {X 0.136,Y -631.180,Z 300.393,A 0.000,B 0.000,C 90.000,E1 286.732} C_DIS
LIN {X 0.176,Y -625.903,Z 300.379,A 0.000,B 0.000,C 90.000,E1 284.189} C_DIS
LIN {X -0.298,Y -621.095,Z 300.363,A 0.000,B 0.000,C 90.000,E1 281.422} C_DIS
LIN {X -0.117,Y -618.052,Z 300.351,A 0.000,B 0.000,C 90.000,E1 279.095} C_DIS
LIN {X 0.093,Y -616.430,Z 300.342,A 0.000,B 0.000,C 90.000,E1 277.530} C_DIS
LIN {X -0.028,Y -614.266,Z 300.326,A 0.000,B 0.000,C 90.000,E1 274.702} C_DIS
LIN {X -0.070,Y -613.388,Z 300.315,A 0.000,B 0.000,C 90.000,E1 272.636} C_DIS
LIN {X -0.153,Y -613.020,Z 300.303,A 0.000,B 0.000,C 90.000,E1 270.573} C_DIS
LIN {X 0.006,Y -613.632,Z 300.284,A 0.000,B 0.000,C 90.000,E1 267.192} C_DIS
LIN {X -0.264,Y -615.839,Z 300.266,A 0.000,B 0.000,C 90.000,E1 263.856} C_DIS
LIN {X 0.197,Y -617.543,Z 300.256,A 0.000,B 0.000,C 90.000,E1 262.008} C_DIS
LIN {X -0.230,Y -621.051,Z 300.240,A 0.000,B 0.000,C 90.000,E1 259.218} C_DIS
LIN {X -0.273,Y -624.052,Z 300.229,A 0.000,B 0.000,C 90.000,E1 257.173} C_DIS
LIN {X -0.311,Y -626.324,Z 300.220,A 0.000,B 0.000,C 90.000,E1 255.644} C_DIS
LIN {X 0.248,Y -627.792,Z 300.214,A 0.000,B 0.000,C 90.000,E1 254.574} C_DIS
LIN {X 0.228,Y -628.937,Z 300.209,A 0.000,B 0.000,C 90.000,E1 253.559} C_DIS
LIN {X 0.022,Y -629.958,Z 300.202,A 0.000,B 0.000,C 90.000,E1 252.308} C_DIS
LIN {X 0.219,Y -630.739,Z 300.196,A 0.000,B 0.000,C 90.000,E1 251.275} C_DIS
LIN {X -0.174,Y -631.043,Z 300.192,A 0.000,B 0.000,C 90.000,E1 250.550} C_DIS
LIN {X 0.038,Y -631.189,Z 300.186,A 0.000,B 0.000,C 90.000,E1 249.518} C_DIS
LIN {X -0.322,Y -630.793,Z 300.179,A 0.000,B 0.000,C 90.000,E1 248.284} C_DIS
LIN {X 0.112,Y -629.952,Z 300.174,A 0.000,B 0.000,C 90.000,E1 247.230} C_DIS
LIN {X -0.067,Y -629.100,Z 300.169,A 0.000,B 0.000,C 90.000,E1 246.485} C_DIS
LIN {X -0.238,Y -627.489,Z 300.164,A 0.000,B 0.000,C 90.000,E1 245.485} C_DIS
